ABB RAPID module: P60.mod

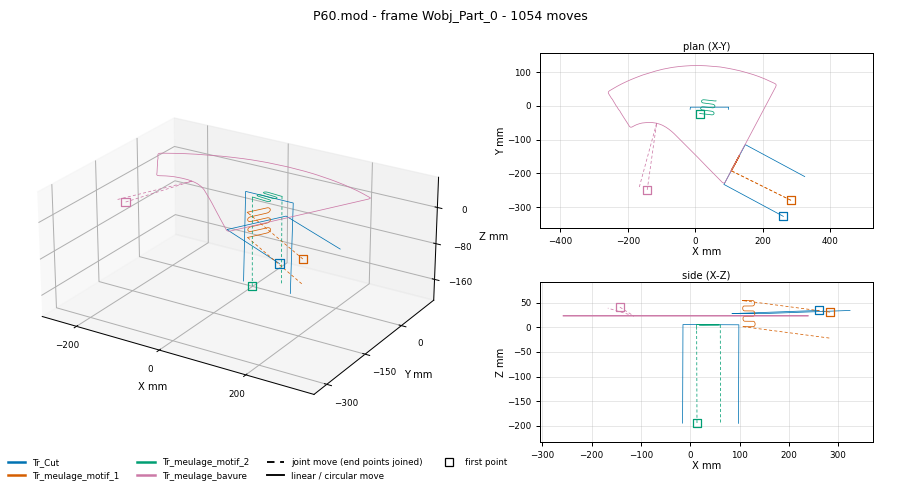
[picture p0: tool path of P60.mod in frame Wobj_Part_0, 1054 of 1064 moves have a stored position in this frame; points joined in program order, loops and branches not executed]
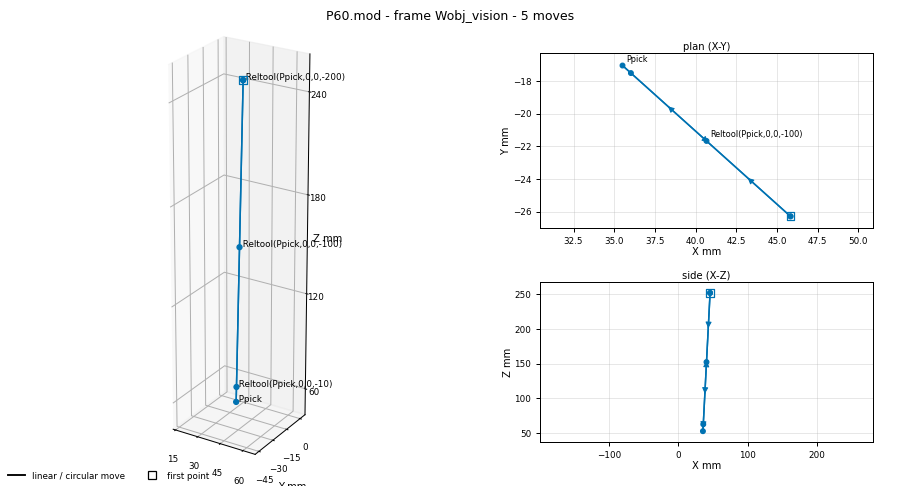
[picture p1: tool path of P60.mod in frame Wobj_vision, 5 of 1064 moves have a stored position in this frame; points joined in program order, loops and branches not executed]
MODULE P60
	LOCAL CONST Speeddata vitesse_Tronconnage :=[10, 500, 0, 0];
	LOCAL CONST Robtarget Coupe_0 :=[[118.6595,-169.366,27.637169921875],[0.183639212461518,0.161711104402732,0.6883672847491,0.682844520843884],[0,0,0,0],[8.999999E+09,8.999999E+09,8.999999E+09,8.999999E+09,8.999999E+09,8.999999E+09]];
	LOCAL CONST Robtarget Coupe_1 :=[[36.94522265625,-3.83223803710937,5.1827177734375],[0.70842525590095,-0.0115011244984384,-0.705597649362176,0.0115472140154091],[0,0,0,0],[8.999999E+09,8.999999E+09,8.999999E+09,8.999999E+09,8.999999E+09,8.999999E+09]];
	LOCAL CONST Robtarget Tr_meulage_motif_1_App1 :=[[283.559670676337,-280.003554022324,30.6185387570368],[0.635107748876336,-0.564376918949611,-0.350307497755773,0.394209966502961],[0,0,0,0],[8.999999E+09,8.999999E+09,8.999999E+09,8.999999E+09,8.999999E+09,8.999999E+09]];
	LOCAL CONST Robtarget Tr_meulage_motif_1_App2 :=[[114.472585877567,-196.272283951116,52.9486118987893],[0.635107748876336,-0.564376918949611,-0.350307497755773,0.394209966502961],[0,0,0,0],[8.999999E+09,8.999999E+09,8.999999E+09,8.999999E+09,8.999999E+09,8.999999E+09]];
	LOCAL CONST Robtarget Tr_meulage_motif_1_P0 :=[[105.573265625,-191.865375,54.12387890625],[0.635107748876336,-0.564376918949611,-0.350307497755773,0.394209966502961],[0,0,0,0],[8.999999E+09,8.999999E+09,8.999999E+09,8.999999E+09,8.999999E+09,8.999999E+09]];
	LOCAL CONST Robtarget Tr_meulage_motif_1_P1 :=[[106.0475625,-190.985015625,54.12386328125],[0.635107748876336,-0.564376918949611,-0.350307497755773,0.394209966502961],[0,0,0,0],[8.999999E+09,8.999999E+09,8.999999E+09,8.999999E+09,8.999999E+09,8.999999E+09]];
	LOCAL CONST Robtarget Tr_meulage_motif_1_P2 :=[[106.5218515625,-190.104640625,54.1238515625],[0.635107748876336,-0.564376918949611,-0.350307497755773,0.394209966502961],[0,0,0,0],[8.999999E+09,8.999999E+09,8.999999E+09,8.999999E+09,8.999999E+09,8.999999E+09]];
	LOCAL CONST Robtarget Tr_meulage_motif_1_P3 :=[[106.9961484375,-189.22428125,54.12383984375],[0.635107748876336,-0.564376918949611,-0.350307497755773,0.394209966502961],[0,0,0,0],[8.999999E+09,8.999999E+09,8.999999E+09,8.999999E+09,8.999999E+09,8.999999E+09]];
	LOCAL CONST Robtarget Tr_meulage_motif_1_P4 :=[[107.4704375,-188.34390625,54.123828125],[0.635107748876336,-0.564376918949611,-0.350307497755773,0.394209966502961],[0,0,0,0],[8.999999E+09,8.999999E+09,8.999999E+09,8.999999E+09,8.999999E+09,8.999999E+09]];
	LOCAL CONST Robtarget Tr_meulage_motif_1_P5 :=[[107.944734375,-187.463546875,54.12381640625],[0.635107748876336,-0.564376918949611,-0.350307497755773,0.394209966502961],[0,0,0,0],[8.999999E+09,8.999999E+09,8.999999E+09,8.999999E+09,8.999999E+09,8.999999E+09]];
	LOCAL CONST Robtarget Tr_meulage_motif_1_P6 :=[[108.4190234375,-186.583171875,54.1238046875],[0.635107748876336,-0.564376918949611,-0.350307497755773,0.394209966502961],[0,0,0,0],[8.999999E+09,8.999999E+09,8.999999E+09,8.999999E+09,8.999999E+09,8.999999E+09]];
	LOCAL CONST Robtarget Tr_meulage_motif_1_P7 :=[[108.8933125,-185.7028125,54.1237890625],[0.635107748876336,-0.564376918949611,-0.350307497755773,0.394209966502961],[0,0,0,0],[8.999999E+09,8.999999E+09,8.999999E+09,8.999999E+09,8.999999E+09,8.999999E+09]];
	LOCAL CONST Robtarget Tr_meulage_motif_1_P8 :=[[109.367609375,-184.8224375,54.12377734375],[0.635107748876336,-0.564376918949611,-0.350307497755773,0.394209966502961],[0,0,0,0],[8.999999E+09,8.999999E+09,8.999999E+09,8.999999E+09,8.999999E+09,8.999999E+09]];
	LOCAL CONST Robtarget Tr_meulage_motif_1_P9 :=[[109.8418984375,-183.942078125,54.123765625],[0.635107748876336,-0.564376918949611,-0.350307497755773,0.394209966502961],[0,0,0,0],[8.999999E+09,8.999999E+09,8.999999E+09,8.999999E+09,8.999999E+09,8.999999E+09]];
	LOCAL CONST Robtarget Tr_meulage_motif_1_P10 :=[[110.3161953125,-183.061703125,54.12375390625],[0.635107748876336,-0.564376918949611,-0.350307497755773,0.394209966502961],[0,0,0,0],[8.999999E+09,8.999999E+09,8.999999E+09,8.999999E+09,8.999999E+09,8.999999E+09]];
	LOCAL CONST Robtarget Tr_meulage_motif_1_P11 :=[[110.790484375,-182.18134375,54.1237421875],[0.635107748876336,-0.564376918949611,-0.350307497755773,0.394209966502961],[0,0,0,0],[8.999999E+09,8.999999E+09,8.999999E+09,8.999999E+09,8.999999E+09,8.999999E+09]];
	LOCAL CONST Robtarget Tr_meulage_motif_1_P12 :=[[111.26478125,-181.30096875,54.1237265625],[0.635107748876336,-0.564376918949611,-0.350307497755773,0.394209966502961],[0,0,0,0],[8.999999E+09,8.999999E+09,8.999999E+09,8.999999E+09,8.999999E+09,8.999999E+09]];
	LOCAL CONST Robtarget Tr_meulage_motif_1_P13 :=[[111.7390703125,-180.420609375,54.12371484375],[0.635107748876336,-0.564376918949611,-0.350307497755773,0.394209966502961],[0,0,0,0],[8.999999E+09,8.999999E+09,8.999999E+09,8.999999E+09,8.999999E+09,8.999999E+09]];
	LOCAL CONST Robtarget Tr_meulage_motif_1_P14 :=[[112.2133671875,-179.540234375,54.123703125],[0.635107748876336,-0.564376918949611,-0.350307497755773,0.394209966502961],[0,0,0,0],[8.999999E+09,8.999999E+09,8.999999E+09,8.999999E+09,8.999999E+09,8.999999E+09]];
	LOCAL CONST Robtarget Tr_meulage_motif_1_P15 :=[[112.68765625,-178.659875,54.12369140625],[0.635107748876336,-0.564376918949611,-0.350307497755773,0.394209966502961],[0,0,0,0],[8.999999E+09,8.999999E+09,8.999999E+09,8.999999E+09,8.999999E+09,8.999999E+09]];
	LOCAL CONST Robtarget Tr_meulage_motif_1_P16 :=[[113.161953125,-177.7795,54.1236796875],[0.635107748876336,-0.564376918949611,-0.350307497755773,0.394209966502961],[0,0,0,0],[8.999999E+09,8.999999E+09,8.999999E+09,8.999999E+09,8.999999E+09,8.999999E+09]];
	LOCAL CONST Robtarget Tr_meulage_motif_1_P17 :=[[113.6362421875,-176.899140625,54.1236640625],[0.635107748876336,-0.564376918949611,-0.350307497755773,0.394209966502961],[0,0,0,0],[8.999999E+09,8.999999E+09,8.999999E+09,8.999999E+09,8.999999E+09,8.999999E+09]];
	LOCAL CONST Robtarget Tr_meulage_motif_1_P18 :=[[114.1105390625,-176.018765625,54.12365234375],[0.635107748876336,-0.564376918949611,-0.350307497755773,0.394209966502961],[0,0,0,0],[8.999999E+09,8.999999E+09,8.999999E+09,8.999999E+09,8.999999E+09,8.999999E+09]];
	LOCAL CONST Robtarget Tr_meulage_motif_1_P19 :=[[114.584828125,-175.13840625,54.123640625],[0.635107748876336,-0.564376918949611,-0.350307497755773,0.394209966502961],[0,0,0,0],[8.999999E+09,8.999999E+09,8.999999E+09,8.999999E+09,8.999999E+09,8.999999E+09]];
	LOCAL CONST Robtarget Tr_meulage_motif_1_P20 :=[[115.059125,-174.25803125,54.12362890625],[0.635107748876336,-0.564376918949611,-0.350307497755773,0.394209966502961],[0,0,0,0],[8.999999E+09,8.999999E+09,8.999999E+09,8.999999E+09,8.999999E+09,8.999999E+09]];
	LOCAL CONST Robtarget Tr_meulage_motif_1_P21 :=[[115.5334140625,-173.377671875,54.1236171875],[0.635107748876336,-0.564376918949611,-0.350307497755773,0.394209966502961],[0,0,0,0],[8.999999E+09,8.999999E+09,8.999999E+09,8.999999E+09,8.999999E+09,8.999999E+09]];
	LOCAL CONST Robtarget Tr_meulage_motif_1_P22 :=[[116.0077109375,-172.497296875,54.12360546875],[0.635107748876336,-0.564376918949611,-0.350307497755773,0.394209966502961],[0,0,0,0],[8.999999E+09,8.999999E+09,8.999999E+09,8.999999E+09,8.999999E+09,8.999999E+09]];
	LOCAL CONST Robtarget Tr_meulage_motif_1_P23 :=[[116.482,-171.6169375,54.12358984375],[0.635107748876336,-0.564376918949611,-0.350307497755773,0.394209966502961],[0,0,0,0],[8.999999E+09,8.999999E+09,8.999999E+09,8.999999E+09,8.999999E+09,8.999999E+09]];
	LOCAL CONST Robtarget Tr_meulage_motif_1_P24 :=[[116.956296875,-170.7365625,54.123578125],[0.635107748876336,-0.564376918949611,-0.350307497755773,0.394209966502961],[0,0,0,0],[8.999999E+09,8.999999E+09,8.999999E+09,8.999999E+09,8.999999E+09,8.999999E+09]];
	LOCAL CONST Robtarget Tr_meulage_motif_1_P25 :=[[117.4305859375,-169.856203125,54.12356640625],[0.635107748876336,-0.564376918949611,-0.350307497755773,0.394209966502961],[0,0,0,0],[8.999999E+09,8.999999E+09,8.999999E+09,8.999999E+09,8.999999E+09,8.999999E+09]];
	LOCAL CONST Robtarget Tr_meulage_motif_1_P26 :=[[117.9048828125,-168.975828125,54.1235546875],[0.635107748876336,-0.564376918949611,-0.350307497755773,0.394209966502961],[0,0,0,0],[8.999999E+09,8.999999E+09,8.999999E+09,8.999999E+09,8.999999E+09,8.999999E+09]];
	LOCAL CONST Robtarget Tr_meulage_motif_1_P27 :=[[118.379171875,-168.09546875,54.12354296875],[0.635107748876336,-0.564376918949611,-0.350307497755773,0.394209966502961],[0,0,0,0],[8.999999E+09,8.999999E+09,8.999999E+09,8.999999E+09,8.999999E+09,8.999999E+09]];
	LOCAL CONST Robtarget Tr_meulage_motif_1_P28 :=[[118.8534609375,-167.21509375,54.12352734375],[0.635107748876336,-0.564376918949611,-0.350307497755773,0.394209966502961],[0,0,0,0],[8.999999E+09,8.999999E+09,8.999999E+09,8.999999E+09,8.999999E+09,8.999999E+09]];
	LOCAL CONST Robtarget Tr_meulage_motif_1_P29 :=[[119.3277578125,-166.334734375,54.123515625],[0.635107748876336,-0.564376918949611,-0.350307497755773,0.394209966502961],[0,0,0,0],[8.999999E+09,8.999999E+09,8.999999E+09,8.999999E+09,8.999999E+09,8.999999E+09]];
	LOCAL CONST Robtarget Tr_meulage_motif_1_P30 :=[[119.802046875,-165.454359375,54.12350390625],[0.635107748876336,-0.564376918949611,-0.350307497755773,0.394209966502961],[0,0,0,0],[8.999999E+09,8.999999E+09,8.999999E+09,8.999999E+09,8.999999E+09,8.999999E+09]];
	LOCAL CONST Robtarget Tr_meulage_motif_1_P31 :=[[120.27634375,-164.574,54.1234921875],[0.635107748876336,-0.564376918949611,-0.350307497755773,0.394209966502961],[0,0,0,0],[8.999999E+09,8.999999E+09,8.999999E+09,8.999999E+09,8.999999E+09,8.999999E+09]];
	LOCAL CONST Robtarget Tr_meulage_motif_1_P32 :=[[120.7506328125,-163.693625,54.12348046875],[0.635107748876336,-0.564376918949611,-0.350307497755773,0.394209966502961],[0,0,0,0],[8.999999E+09,8.999999E+09,8.999999E+09,8.999999E+09,8.999999E+09,8.999999E+09]];
	LOCAL CONST Robtarget Tr_meulage_motif_1_P33 :=[[121.2249296875,-162.813265625,54.12346484375],[0.635107748876336,-0.564376918949611,-0.350307497755773,0.394209966502961],[0,0,0,0],[8.999999E+09,8.999999E+09,8.999999E+09,8.999999E+09,8.999999E+09,8.999999E+09]];
	LOCAL CONST Robtarget Tr_meulage_motif_1_P34 :=[[121.69921875,-161.932890625,54.123453125],[0.635107748876336,-0.564376918949611,-0.350307497755773,0.394209966502961],[0,0,0,0],[8.999999E+09,8.999999E+09,8.999999E+09,8.999999E+09,8.999999E+09,8.999999E+09]];
	LOCAL CONST Robtarget Tr_meulage_motif_1_P35 :=[[122.173515625,-161.05253125,54.12344140625],[0.635107748876336,-0.564376918949611,-0.350307497755773,0.394209966502961],[0,0,0,0],[8.999999E+09,8.999999E+09,8.999999E+09,8.999999E+09,8.999999E+09,8.999999E+09]];
	LOCAL CONST Robtarget Tr_meulage_motif_1_P36 :=[[122.6478046875,-160.17215625,54.1234296875],[0.635107748876336,-0.564376918949611,-0.350307497755773,0.394209966502961],[0,0,0,0],[8.999999E+09,8.999999E+09,8.999999E+09,8.999999E+09,8.999999E+09,8.999999E+09]];
	LOCAL CONST Robtarget Tr_meulage_motif_1_P37 :=[[123.1221015625,-159.291796875,54.12341796875],[0.635107748876336,-0.564376918949611,-0.350307497755773,0.394209966502961],[0,0,0,0],[8.999999E+09,8.999999E+09,8.999999E+09,8.999999E+09,8.999999E+09,8.999999E+09]];
	LOCAL CONST Robtarget Tr_meulage_motif_1_P38 :=[[123.596390625,-158.411421875,54.12340625],[0.635107748876336,-0.564376918949611,-0.350307497755773,0.394209966502961],[0,0,0,0],[8.999999E+09,8.999999E+09,8.999999E+09,8.999999E+09,8.999999E+09,8.999999E+09]];
	LOCAL CONST Robtarget Tr_meulage_motif_1_P39 :=[[124.0706875,-157.5310625,54.123390625],[0.635107748876336,-0.564376918949611,-0.350307497755773,0.394209966502961],[0,0,0,0],[8.999999E+09,8.999999E+09,8.999999E+09,8.999999E+09,8.999999E+09,8.999999E+09]];
	LOCAL CONST Robtarget Tr_meulage_motif_1_P40 :=[[124.5449765625,-156.6506875,54.12337890625],[0.635107748876336,-0.564376918949611,-0.350307497755773,0.394209966502961],[0,0,0,0],[8.999999E+09,8.999999E+09,8.999999E+09,8.999999E+09,8.999999E+09,8.999999E+09]];
	LOCAL CONST Robtarget Tr_meulage_motif_1_P41 :=[[125.0192734375,-155.770328125,54.1233671875],[0.635107748876336,-0.564376918949611,-0.350307497755773,0.394209966502961],[0,0,0,0],[8.999999E+09,8.999999E+09,8.999999E+09,8.999999E+09,8.999999E+09,8.999999E+09]];
	LOCAL CONST Robtarget Tr_meulage_motif_1_P42 :=[[125.4935625,-154.889953125,54.12335546875],[0.635107748876336,-0.564376918949611,-0.350307497755773,0.394209966502961],[0,0,0,0],[8.999999E+09,8.999999E+09,8.999999E+09,8.999999E+09,8.999999E+09,8.999999E+09]];
	LOCAL CONST Robtarget Tr_meulage_motif_1_P43 :=[[125.967859375,-154.00959375,54.12334375],[0.635107748876336,-0.564376918949611,-0.350307497755773,0.394209966502961],[0,0,0,0],[8.999999E+09,8.999999E+09,8.999999E+09,8.999999E+09,8.999999E+09,8.999999E+09]];
	LOCAL CONST Robtarget Tr_meulage_motif_1_P44 :=[[126.4421484375,-153.12921875,54.123328125],[0.635107748876336,-0.564376918949611,-0.350307497755773,0.394209966502961],[0,0,0,0],[8.999999E+09,8.999999E+09,8.999999E+09,8.999999E+09,8.999999E+09,8.999999E+09]];
	LOCAL CONST Robtarget Tr_meulage_motif_1_P45 :=[[126.9164453125,-152.248859375,54.12331640625],[0.635107748876336,-0.564376918949611,-0.350307497755773,0.394209966502961],[0,0,0,0],[8.999999E+09,8.999999E+09,8.999999E+09,8.999999E+09,8.999999E+09,8.999999E+09]];
	LOCAL CONST Robtarget Tr_meulage_motif_1_P46 :=[[127.390328125,-151.37671875,54.01276953125],[0.635107748876336,-0.564376918949611,-0.350307497755773,0.394209966502961],[0,0,0,0],[8.999999E+09,8.999999E+09,8.999999E+09,8.999999E+09,8.999999E+09,8.999999E+09]];
	LOCAL CONST Robtarget Tr_meulage_motif_1_P47 :=[[127.845203125,-150.546671875,53.80167578125],[0.635107748876336,-0.564376918949611,-0.350307497755773,0.394209966502961],[0,0,0,0],[8.999999E+09,8.999999E+09,8.999999E+09,8.999999E+09,8.999999E+09,8.999999E+09]];
	LOCAL CONST Robtarget Tr_meulage_motif_1_P48 :=[[128.2573125,-149.80009375,53.5299609375],[0.635107748876336,-0.564376918949611,-0.350307497755773,0.394209966502961],[0,0,0,0],[8.999999E+09,8.999999E+09,8.999999E+09,8.999999E+09,8.999999E+09,8.999999E+09]];
	LOCAL CONST Robtarget Tr_meulage_motif_1_P49 :=[[128.6207890625,-149.144078125,53.25415625],[0.635107748876336,-0.564376918949611,-0.350307497755773,0.394209966502961],[0,0,0,0],[8.999999E+09,8.999999E+09,8.999999E+09,8.999999E+09,8.999999E+09,8.999999E+09]];
	LOCAL CONST Robtarget Tr_meulage_motif_1_P50 :=[[129.160390625,-148.184109375,52.6383359375],[0.635107748876336,-0.564376918949611,-0.350307497755773,0.394209966502961],[0,0,0,0],[8.999999E+09,8.999999E+09,8.999999E+09,8.999999E+09,8.999999E+09,8.999999E+09]];
	LOCAL CONST Robtarget Tr_meulage_motif_1_P51 :=[[129.669921875,-147.295609375,51.7911015625],[0.635107748876336,-0.564376918949611,-0.350307497755773,0.394209966502961],[0,0,0,0],[8.999999E+09,8.999999E+09,8.999999E+09,8.999999E+09,8.999999E+09,8.999999E+09]];
	LOCAL CONST Robtarget Tr_meulage_motif_1_P52 :=[[130.1008515625,-146.5649375,50.7677421875],[0.635107748876336,-0.564376918949611,-0.350307497755773,0.394209966502961],[0,0,0,0],[8.999999E+09,8.999999E+09,8.999999E+09,8.999999E+09,8.999999E+09,8.999999E+09]];
	LOCAL CONST Robtarget Tr_meulage_motif_1_P53 :=[[130.3638671875,-146.152171875,49.65212109375],[0.635107748876336,-0.564376918949611,-0.350307497755773,0.394209966502961],[0,0,0,0],[8.999999E+09,8.999999E+09,8.999999E+09,8.999999E+09,8.999999E+09,8.999999E+09]];
	LOCAL CONST Robtarget Tr_meulage_motif_1_P54 :=[[130.3963359375,-146.1389375,48.95651171875],[0.635107748876336,-0.564376918949611,-0.350307497755773,0.394209966502961],[0,0,0,0],[8.999999E+09,8.999999E+09,8.999999E+09,8.999999E+09,8.999999E+09,8.999999E+09]];
	LOCAL CONST Robtarget Tr_meulage_motif_1_P55 :=[[130.4149921875,-146.148984375,48.2956015625],[0.635107748876336,-0.564376918949611,-0.350307497755773,0.394209966502961],[0,0,0,0],[8.999999E+09,8.999999E+09,8.999999E+09,8.999999E+09,8.999999E+09,8.999999E+09]];
	LOCAL CONST Robtarget Tr_meulage_motif_1_P56 :=[[130.4076171875,-146.207359375,47.63484765625],[0.635107748876336,-0.564376918949611,-0.350307497755773,0.394209966502961],[0,0,0,0],[8.999999E+09,8.999999E+09,8.999999E+09,8.999999E+09,8.999999E+09,8.999999E+09]];
	LOCAL CONST Robtarget Tr_meulage_motif_1_P57 :=[[130.2023984375,-146.662734375,46.53366796875],[0.635107748876336,-0.564376918949611,-0.350307497755773,0.394209966502961],[0,0,0,0],[8.999999E+09,8.999999E+09,8.999999E+09,8.999999E+09,8.999999E+09,8.999999E+09]];
	LOCAL CONST Robtarget Tr_meulage_motif_1_P58 :=[[129.8245078125,-147.4321875,45.52757421875],[0.635107748876336,-0.564376918949611,-0.350307497755773,0.394209966502961],[0,0,0,0],[8.999999E+09,8.999999E+09,8.999999E+09,8.999999E+09,8.999999E+09,8.999999E+09]];
	LOCAL CONST Robtarget Tr_meulage_motif_1_P59 :=[[129.3625,-148.34578125,44.69913671875],[0.635107748876336,-0.564376918949611,-0.350307497755773,0.394209966502961],[0,0,0,0],[8.999999E+09,8.999999E+09,8.999999E+09,8.999999E+09,8.999999E+09,8.999999E+09]];
	LOCAL CONST Robtarget Tr_meulage_motif_1_P60 :=[[129.04778125,-148.9566875,44.30359765625],[0.635107748876336,-0.564376918949611,-0.350307497755773,0.394209966502961],[0,0,0,0],[8.999999E+09,8.999999E+09,8.999999E+09,8.999999E+09,8.999999E+09,8.999999E+09]];
	LOCAL CONST Robtarget Tr_meulage_motif_1_P61 :=[[128.5122265625,-149.98371875,43.81633203125],[0.635107748876336,-0.564376918949611,-0.350307497755773,0.394209966502961],[0,0,0,0],[8.999999E+09,8.999999E+09,8.999999E+09,8.999999E+09,8.999999E+09,8.999999E+09]];
	LOCAL CONST Robtarget Tr_meulage_motif_1_P62 :=[[128.1188828125,-150.731671875,43.5523828125],[0.635107748876336,-0.564376918949611,-0.350307497755773,0.394209966502961],[0,0,0,0],[8.999999E+09,8.999999E+09,8.999999E+09,8.999999E+09,8.999999E+09,8.999999E+09]];
	LOCAL CONST Robtarget Tr_meulage_motif_1_P63 :=[[127.6826171875,-151.55528125,43.34803125],[0.635107748876336,-0.564376918949611,-0.350307497755773,0.394209966502961],[0,0,0,0],[8.999999E+09,8.999999E+09,8.999999E+09,8.999999E+09,8.999999E+09,8.999999E+09]];
	LOCAL CONST Robtarget Tr_meulage_motif_1_P64 :=[[127.2201328125,-152.4210625,43.2395078125],[0.635107748876336,-0.564376918949611,-0.350307497755773,0.394209966502961],[0,0,0,0],[8.999999E+09,8.999999E+09,8.999999E+09,8.999999E+09,8.999999E+09,8.999999E+09]];
	LOCAL CONST Robtarget Tr_meulage_motif_1_P65 :=[[126.752484375,-153.2965625,43.12898046875],[0.635107748876336,-0.564376918949611,-0.350307497755773,0.394209966502961],[0,0,0,0],[8.999999E+09,8.999999E+09,8.999999E+09,8.999999E+09,8.999999E+09,8.999999E+09]];
	LOCAL CONST Robtarget Tr_meulage_motif_1_P66 :=[[126.2781875,-154.1769375,43.12899609375],[0.635107748876336,-0.564376918949611,-0.350307497755773,0.394209966502961],[0,0,0,0],[8.999999E+09,8.999999E+09,8.999999E+09,8.999999E+09,8.999999E+09,8.999999E+09]];
	LOCAL CONST Robtarget Tr_meulage_motif_1_P67 :=[[125.8038984375,-155.057296875,43.1290078125],[0.635107748876336,-0.564376918949611,-0.350307497755773,0.394209966502961],[0,0,0,0],[8.999999E+09,8.999999E+09,8.999999E+09,8.999999E+09,8.999999E+09,8.999999E+09]];
	LOCAL CONST Robtarget Tr_meulage_motif_1_P68 :=[[125.329609375,-155.937671875,43.12901953125],[0.635107748876336,-0.564376918949611,-0.350307497755773,0.394209966502961],[0,0,0,0],[8.999999E+09,8.999999E+09,8.999999E+09,8.999999E+09,8.999999E+09,8.999999E+09]];
	LOCAL CONST Robtarget Tr_meulage_motif_1_P69 :=[[124.8553125,-156.81803125,43.12903125],[0.635107748876336,-0.564376918949611,-0.350307497755773,0.394209966502961],[0,0,0,0],[8.999999E+09,8.999999E+09,8.999999E+09,8.999999E+09,8.999999E+09,8.999999E+09]];
	LOCAL CONST Robtarget Tr_meulage_motif_1_P70 :=[[124.3810234375,-157.69840625,43.12904296875],[0.635107748876336,-0.564376918949611,-0.350307497755773,0.394209966502961],[0,0,0,0],[8.999999E+09,8.999999E+09,8.999999E+09,8.999999E+09,8.999999E+09,8.999999E+09]];
	LOCAL CONST Robtarget Tr_meulage_motif_1_P71 :=[[123.9067265625,-158.578765625,43.1290546875],[0.635107748876336,-0.564376918949611,-0.350307497755773,0.394209966502961],[0,0,0,0],[8.999999E+09,8.999999E+09,8.999999E+09,8.999999E+09,8.999999E+09,8.999999E+09]];
	LOCAL CONST Robtarget Tr_meulage_motif_1_P72 :=[[123.4324375,-159.459140625,43.1290703125],[0.635107748876336,-0.564376918949611,-0.350307497755773,0.394209966502961],[0,0,0,0],[8.999999E+09,8.999999E+09,8.999999E+09,8.999999E+09,8.999999E+09,8.999999E+09]];
	LOCAL CONST Robtarget Tr_meulage_motif_1_P73 :=[[122.958140625,-160.3395,43.12908203125],[0.635107748876336,-0.564376918949611,-0.350307497755773,0.394209966502961],[0,0,0,0],[8.999999E+09,8.999999E+09,8.999999E+09,8.999999E+09,8.999999E+09,8.999999E+09]];
	LOCAL CONST Robtarget Tr_meulage_motif_1_P74 :=[[122.4838515625,-161.219875,43.12909375],[0.635107748876336,-0.564376918949611,-0.350307497755773,0.394209966502961],[0,0,0,0],[8.999999E+09,8.999999E+09,8.999999E+09,8.999999E+09,8.999999E+09,8.999999E+09]];
	LOCAL CONST Robtarget Tr_meulage_motif_1_P75 :=[[122.0095546875,-162.100234375,43.12910546875],[0.635107748876336,-0.564376918949611,-0.350307497755773,0.394209966502961],[0,0,0,0],[8.999999E+09,8.999999E+09,8.999999E+09,8.999999E+09,8.999999E+09,8.999999E+09]];
	LOCAL CONST Robtarget Tr_meulage_motif_1_P76 :=[[121.535265625,-162.980609375,43.1291171875],[0.635107748876336,-0.564376918949611,-0.350307497755773,0.394209966502961],[0,0,0,0],[8.999999E+09,8.999999E+09,8.999999E+09,8.999999E+09,8.999999E+09,8.999999E+09]];
	LOCAL CONST Robtarget Tr_meulage_motif_1_P77 :=[[121.06096875,-163.86096875,43.1291328125],[0.635107748876336,-0.564376918949611,-0.350307497755773,0.394209966502961],[0,0,0,0],[8.999999E+09,8.999999E+09,8.999999E+09,8.999999E+09,8.999999E+09,8.999999E+09]];
	LOCAL CONST Robtarget Tr_meulage_motif_1_P78 :=[[120.5866796875,-164.74134375,43.12914453125],[0.635107748876336,-0.564376918949611,-0.350307497755773,0.394209966502961],[0,0,0,0],[8.999999E+09,8.999999E+09,8.999999E+09,8.999999E+09,8.999999E+09,8.999999E+09]];
	LOCAL CONST Robtarget Tr_meulage_motif_1_P79 :=[[120.1123828125,-165.621703125,43.12915625],[0.635107748876336,-0.564376918949611,-0.350307497755773,0.394209966502961],[0,0,0,0],[8.999999E+09,8.999999E+09,8.999999E+09,8.999999E+09,8.999999E+09,8.999999E+09]];
	LOCAL CONST Robtarget Tr_meulage_motif_1_P80 :=[[119.63809375,-166.502078125,43.12916796875],[0.635107748876336,-0.564376918949611,-0.350307497755773,0.394209966502961],[0,0,0,0],[8.999999E+09,8.999999E+09,8.999999E+09,8.999999E+09,8.999999E+09,8.999999E+09]];
	LOCAL CONST Robtarget Tr_meulage_motif_1_P81 :=[[119.163796875,-167.3824375,43.1291796875],[0.635107748876336,-0.564376918949611,-0.350307497755773,0.394209966502961],[0,0,0,0],[8.999999E+09,8.999999E+09,8.999999E+09,8.999999E+09,8.999999E+09,8.999999E+09]];
	LOCAL CONST Robtarget Tr_meulage_motif_1_P82 :=[[118.6895078125,-168.2628125,43.1291953125],[0.635107748876336,-0.564376918949611,-0.350307497755773,0.394209966502961],[0,0,0,0],[8.999999E+09,8.999999E+09,8.999999E+09,8.999999E+09,8.999999E+09,8.999999E+09]];
	LOCAL CONST Robtarget Tr_meulage_motif_1_P83 :=[[118.2152109375,-169.143171875,43.12920703125],[0.635107748876336,-0.564376918949611,-0.350307497755773,0.394209966502961],[0,0,0,0],[8.999999E+09,8.999999E+09,8.999999E+09,8.999999E+09,8.999999E+09,8.999999E+09]];
	LOCAL CONST Robtarget Tr_meulage_motif_1_P84 :=[[117.740921875,-170.023546875,43.12921875],[0.635107748876336,-0.564376918949611,-0.350307497755773,0.394209966502961],[0,0,0,0],[8.999999E+09,8.999999E+09,8.999999E+09,8.999999E+09,8.999999E+09,8.999999E+09]];
	LOCAL CONST Robtarget Tr_meulage_motif_1_P85 :=[[117.266625,-170.90390625,43.12923046875],[0.635107748876336,-0.564376918949611,-0.350307497755773,0.394209966502961],[0,0,0,0],[8.999999E+09,8.999999E+09,8.999999E+09,8.999999E+09,8.999999E+09,8.999999E+09]];
	LOCAL CONST Robtarget Tr_meulage_motif_1_P86 :=[[116.7923359375,-171.78428125,43.1292421875],[0.635107748876336,-0.564376918949611,-0.350307497755773,0.394209966502961],[0,0,0,0],[8.999999E+09,8.999999E+09,8.999999E+09,8.999999E+09,8.999999E+09,8.999999E+09]];
	LOCAL CONST Robtarget Tr_meulage_motif_1_P87 :=[[116.3180390625,-172.664640625,43.12925390625],[0.635107748876336,-0.564376918949611,-0.350307497755773,0.394209966502961],[0,0,0,0],[8.999999E+09,8.999999E+09,8.999999E+09,8.999999E+09,8.999999E+09,8.999999E+09]];
	LOCAL CONST Robtarget Tr_meulage_motif_1_P88 :=[[115.84375,-173.545015625,43.12926953125],[0.635107748876336,-0.564376918949611,-0.350307497755773,0.394209966502961],[0,0,0,0],[8.999999E+09,8.999999E+09,8.999999E+09,8.999999E+09,8.999999E+09,8.999999E+09]];
	LOCAL CONST Robtarget Tr_meulage_motif_1_P89 :=[[115.3694609375,-174.425375,43.12928125],[0.635107748876336,-0.564376918949611,-0.350307497755773,0.394209966502961],[0,0,0,0],[8.999999E+09,8.999999E+09,8.999999E+09,8.999999E+09,8.999999E+09,8.999999E+09]];
	LOCAL CONST Robtarget Tr_meulage_motif_1_P90 :=[[114.8951640625,-175.30575,43.12929296875],[0.635107748876336,-0.564376918949611,-0.350307497755773,0.394209966502961],[0,0,0,0],[8.999999E+09,8.999999E+09,8.999999E+09,8.999999E+09,8.999999E+09,8.999999E+09]];
	LOCAL CONST Robtarget Tr_meulage_motif_1_P91 :=[[114.420875,-176.186109375,43.1293046875],[0.635107748876336,-0.564376918949611,-0.350307497755773,0.394209966502961],[0,0,0,0],[8.999999E+09,8.999999E+09,8.999999E+09,8.999999E+09,8.999999E+09,8.999999E+09]];
	LOCAL CONST Robtarget Tr_meulage_motif_1_P92 :=[[113.946578125,-177.066484375,43.12931640625],[0.635107748876336,-0.564376918949611,-0.350307497755773,0.394209966502961],[0,0,0,0],[8.999999E+09,8.999999E+09,8.999999E+09,8.999999E+09,8.999999E+09,8.999999E+09]];
	LOCAL CONST Robtarget Tr_meulage_motif_1_P93 :=[[113.4722890625,-177.94684375,43.12933203125],[0.635107748876336,-0.564376918949611,-0.350307497755773,0.394209966502961],[0,0,0,0],[8.999999E+09,8.999999E+09,8.999999E+09,8.999999E+09,8.999999E+09,8.999999E+09]];
	LOCAL CONST Robtarget Tr_meulage_motif_1_P94 :=[[112.9979921875,-178.82721875,43.12934375],[0.635107748876336,-0.564376918949611,-0.350307497755773,0.394209966502961],[0,0,0,0],[8.999999E+09,8.999999E+09,8.999999E+09,8.999999E+09,8.999999E+09,8.999999E+09]];
	LOCAL CONST Robtarget Tr_meulage_motif_1_P95 :=[[112.523703125,-179.707578125,43.12935546875],[0.635107748876336,-0.564376918949611,-0.350307497755773,0.394209966502961],[0,0,0,0],[8.999999E+09,8.999999E+09,8.999999E+09,8.999999E+09,8.999999E+09,8.999999E+09]];
	LOCAL CONST Robtarget Tr_meulage_motif_1_P96 :=[[112.04940625,-180.587953125,43.1293671875],[0.635107748876336,-0.564376918949611,-0.350307497755773,0.394209966502961],[0,0,0,0],[8.999999E+09,8.999999E+09,8.999999E+09,8.999999E+09,8.999999E+09,8.999999E+09]];
	LOCAL CONST Robtarget Tr_meulage_motif_1_P97 :=[[111.5751171875,-181.4683125,43.12937890625],[0.635107748876336,-0.564376918949611,-0.350307497755773,0.394209966502961],[0,0,0,0],[8.999999E+09,8.999999E+09,8.999999E+09,8.999999E+09,8.999999E+09,8.999999E+09]];
	LOCAL CONST Robtarget Tr_meulage_motif_1_P98 :=[[111.1008203125,-182.3486875,43.12939453125],[0.635107748876336,-0.564376918949611,-0.350307497755773,0.394209966502961],[0,0,0,0],[8.999999E+09,8.999999E+09,8.999999E+09,8.999999E+09,8.999999E+09,8.999999E+09]];
	LOCAL CONST Robtarget Tr_meulage_motif_1_P99 :=[[110.62653125,-183.229046875,43.12940625],[0.635107748876336,-0.564376918949611,-0.350307497755773,0.394209966502961],[0,0,0,0],[8.999999E+09,8.999999E+09,8.999999E+09,8.999999E+09,8.999999E+09,8.999999E+09]];
	LOCAL CONST Robtarget Tr_meulage_motif_1_P100 :=[[110.152234375,-184.109421875,43.12941796875],[0.635107748876336,-0.564376918949611,-0.350307497755773,0.394209966502961],[0,0,0,0],[8.999999E+09,8.999999E+09,8.999999E+09,8.999999E+09,8.999999E+09,8.999999E+09]];
	LOCAL CONST Robtarget Tr_meulage_motif_1_P101 :=[[109.6779453125,-184.98978125,43.1294296875],[0.635107748876336,-0.564376918949611,-0.350307497755773,0.394209966502961],[0,0,0,0],[8.999999E+09,8.999999E+09,8.999999E+09,8.999999E+09,8.999999E+09,8.999999E+09]];
	LOCAL CONST Robtarget Tr_meulage_motif_1_P102 :=[[109.2036484375,-185.87015625,43.12944140625],[0.635107748876336,-0.564376918949611,-0.350307497755773,0.394209966502961],[0,0,0,0],[8.999999E+09,8.999999E+09,8.999999E+09,8.999999E+09,8.999999E+09,8.999999E+09]];
	LOCAL CONST Robtarget Tr_meulage_motif_1_P103 :=[[108.7360078125,-186.74565625,43.01891796875],[0.635107748876336,-0.564376918949611,-0.350307497755773,0.394209966502961],[0,0,0,0],[8.999999E+09,8.999999E+09,8.999999E+09,8.999999E+09,8.999999E+09,8.999999E+09]];
	LOCAL CONST Robtarget Tr_meulage_motif_1_P104 :=[[108.293046875,-187.582140625,42.8078515625],[0.635107748876336,-0.564376918949611,-0.350307497755773,0.394209966502961],[0,0,0,0],[8.999999E+09,8.999999E+09,8.999999E+09,8.999999E+09,8.999999E+09,8.999999E+09]];
	LOCAL CONST Robtarget Tr_meulage_motif_1_P105 :=[[107.8962734375,-188.336984375,42.53615625],[0.635107748876336,-0.564376918949611,-0.350307497755773,0.394209966502961],[0,0,0,0],[8.999999E+09,8.999999E+09,8.999999E+09,8.999999E+09,8.999999E+09,8.999999E+09]];
	LOCAL CONST Robtarget Tr_meulage_motif_1_P106 :=[[107.5673984375,-188.967984375,42.23216796875],[0.635107748876336,-0.564376918949611,-0.350307497755773,0.394209966502961],[0,0,0,0],[8.999999E+09,8.999999E+09,8.999999E+09,8.999999E+09,8.999999E+09,8.999999E+09]];
	LOCAL CONST Robtarget Tr_meulage_motif_1_P107 :=[[107.0954453125,-189.88878125,41.56998828125],[0.635107748876336,-0.564376918949611,-0.350307497755773,0.394209966502961],[0,0,0,0],[8.999999E+09,8.999999E+09,8.999999E+09,8.999999E+09,8.999999E+09,8.999999E+09]];
	LOCAL CONST Robtarget Tr_meulage_motif_1_P108 :=[[106.693109375,-190.69653125,40.6685234375],[0.635107748876336,-0.564376918949611,-0.350307497755773,0.394209966502961],[0,0,0,0],[8.999999E+09,8.999999E+09,8.999999E+09,8.999999E+09,8.999999E+09,8.999999E+09]];
	LOCAL CONST Robtarget Tr_meulage_motif_1_P109 :=[[106.468890625,-191.183421875,39.6230390625],[0.635107748876336,-0.564376918949611,-0.350307497755773,0.394209966502961],[0,0,0,0],[8.999999E+09,8.999999E+09,8.999999E+09,8.999999E+09,8.999999E+09,8.999999E+09]];
	LOCAL CONST Robtarget Tr_meulage_motif_1_P110 :=[[106.4008046875,-191.356640625,38.9301796875],[0.635107748876336,-0.564376918949611,-0.350307497755773,0.394209966502961],[0,0,0,0],[8.999999E+09,8.999999E+09,8.999999E+09,8.999999E+09,8.999999E+09,8.999999E+09]];
	LOCAL CONST Robtarget Tr_meulage_motif_1_P111 :=[[106.39225,-191.4245625,38.16057421875],[0.635107748876336,-0.564376918949611,-0.350307497755773,0.394209966502961],[0,0,0,0],[8.999999E+09,8.999999E+09,8.999999E+09,8.999999E+09,8.999999E+09,8.999999E+09]];
	LOCAL CONST Robtarget Tr_meulage_motif_1_P112 :=[[106.44571875,-191.37734375,37.39109375],[0.635107748876336,-0.564376918949611,-0.350307497755773,0.394209966502961],[0,0,0,0],[8.999999E+09,8.999999E+09,8.999999E+09,8.999999E+09,8.999999E+09,8.999999E+09]];
	LOCAL CONST Robtarget Tr_meulage_motif_1_P113 :=[[106.6759921875,-191.0248125,36.28341015625],[0.635107748876336,-0.564376918949611,-0.350307497755773,0.394209966502961],[0,0,0,0],[8.999999E+09,8.999999E+09,8.999999E+09,8.999999E+09,8.999999E+09,8.999999E+09]];
	LOCAL CONST Robtarget Tr_meulage_motif_1_P114 :=[[106.8890234375,-190.66896875,35.698015625],[0.635107748876336,-0.564376918949611,-0.350307497755773,0.394209966502961],[0,0,0,0],[8.999999E+09,8.999999E+09,8.999999E+09,8.999999E+09,8.999999E+09,8.999999E+09]];
	LOCAL CONST Robtarget Tr_meulage_motif_1_P115 :=[[107.3348125,-189.90146875,34.8113359375],[0.635107748876336,-0.564376918949611,-0.350307497755773,0.394209966502961],[0,0,0,0],[8.999999E+09,8.999999E+09,8.999999E+09,8.999999E+09,8.999999E+09,8.999999E+09]];
	LOCAL CONST Robtarget Tr_meulage_motif_1_P116 :=[[107.6242890625,-189.39215625,34.39723046875],[0.635107748876336,-0.564376918949611,-0.350307497755773,0.394209966502961],[0,0,0,0],[8.999999E+09,8.999999E+09,8.999999E+09,8.999999E+09,8.999999E+09,8.999999E+09]];
	LOCAL CONST Robtarget Tr_meulage_motif_1_P117 :=[[108.1698515625,-188.416265625,33.85340234375],[0.635107748876336,-0.564376918949611,-0.350307497755773,0.394209966502961],[0,0,0,0],[8.999999E+09,8.999999E+09,8.999999E+09,8.999999E+09,8.999999E+09,8.999999E+09]];
	LOCAL CONST Robtarget Tr_meulage_motif_1_P118 :=[[108.5697578125,-187.6939375,33.55804296875],[0.635107748876336,-0.564376918949611,-0.350307497755773,0.394209966502961],[0,0,0,0],[8.999999E+09,8.999999E+09,8.999999E+09,8.999999E+09,8.999999E+09,8.999999E+09]];
	LOCAL CONST Robtarget Tr_meulage_motif_1_P119 :=[[109.0175703125,-186.876546875,33.35366796875],[0.635107748876336,-0.564376918949611,-0.350307497755773,0.394209966502961],[0,0,0,0],[8.999999E+09,8.999999E+09,8.999999E+09,8.999999E+09,8.999999E+09,8.999999E+09]];
	LOCAL CONST Robtarget Tr_meulage_motif_1_P120 :=[[109.4861796875,-186.0140625,33.2451171875],[0.635107748876336,-0.564376918949611,-0.350307497755773,0.394209966502961],[0,0,0,0],[8.999999E+09,8.999999E+09,8.999999E+09,8.999999E+09,8.999999E+09,8.999999E+09]];
	LOCAL CONST Robtarget Tr_meulage_motif_1_P121 :=[[109.9600703125,-185.141921875,33.13456640625],[0.635107748876336,-0.564376918949611,-0.350307497755773,0.394209966502961],[0,0,0,0],[8.999999E+09,8.999999E+09,8.999999E+09,8.999999E+09,8.999999E+09,8.999999E+09]];
	LOCAL CONST Robtarget Tr_meulage_motif_1_P122 :=[[110.434359375,-184.261546875,33.1345546875],[0.635107748876336,-0.564376918949611,-0.350307497755773,0.394209966502961],[0,0,0,0],[8.999999E+09,8.999999E+09,8.999999E+09,8.999999E+09,8.999999E+09,8.999999E+09]];
	LOCAL CONST Robtarget Tr_meulage_motif_1_P123 :=[[110.9086484375,-183.3811875,33.13454296875],[0.635107748876336,-0.564376918949611,-0.350307497755773,0.394209966502961],[0,0,0,0],[8.999999E+09,8.999999E+09,8.999999E+09,8.999999E+09,8.999999E+09,8.999999E+09]];
	LOCAL CONST Robtarget Tr_meulage_motif_1_P124 :=[[111.3829453125,-182.5008125,33.13453125],[0.635107748876336,-0.564376918949611,-0.350307497755773,0.394209966502961],[0,0,0,0],[8.999999E+09,8.999999E+09,8.999999E+09,8.999999E+09,8.999999E+09,8.999999E+09]];
	LOCAL CONST Robtarget Tr_meulage_motif_1_P125 :=[[111.857234375,-181.620453125,33.13451953125],[0.635107748876336,-0.564376918949611,-0.350307497755773,0.394209966502961],[0,0,0,0],[8.999999E+09,8.999999E+09,8.999999E+09,8.999999E+09,8.999999E+09,8.999999E+09]];
	LOCAL CONST Robtarget Tr_meulage_motif_1_P126 :=[[112.33153125,-180.740078125,33.1345078125],[0.635107748876336,-0.564376918949611,-0.350307497755773,0.394209966502961],[0,0,0,0],[8.999999E+09,8.999999E+09,8.999999E+09,8.999999E+09,8.999999E+09,8.999999E+09]];
	LOCAL CONST Robtarget Tr_meulage_motif_1_P127 :=[[112.8058203125,-179.85971875,33.1344921875],[0.635107748876336,-0.564376918949611,-0.350307497755773,0.394209966502961],[0,0,0,0],[8.999999E+09,8.999999E+09,8.999999E+09,8.999999E+09,8.999999E+09,8.999999E+09]];
	LOCAL CONST Robtarget Tr_meulage_motif_1_P128 :=[[113.2801171875,-178.97934375,33.13448046875],[0.635107748876336,-0.564376918949611,-0.350307497755773,0.394209966502961],[0,0,0,0],[8.999999E+09,8.999999E+09,8.999999E+09,8.999999E+09,8.999999E+09,8.999999E+09]];
	LOCAL CONST Robtarget Tr_meulage_motif_1_P129 :=[[113.75440625,-178.098984375,33.13446875],[0.635107748876336,-0.564376918949611,-0.350307497755773,0.394209966502961],[0,0,0,0],[8.999999E+09,8.999999E+09,8.999999E+09,8.999999E+09,8.999999E+09,8.999999E+09]];
	LOCAL CONST Robtarget Tr_meulage_motif_1_P130 :=[[114.228703125,-177.218609375,33.13445703125],[0.635107748876336,-0.564376918949611,-0.350307497755773,0.394209966502961],[0,0,0,0],[8.999999E+09,8.999999E+09,8.999999E+09,8.999999E+09,8.999999E+09,8.999999E+09]];
	LOCAL CONST Robtarget Tr_meulage_motif_1_P131 :=[[114.7029921875,-176.33825,33.1344453125],[0.635107748876336,-0.564376918949611,-0.350307497755773,0.394209966502961],[0,0,0,0],[8.999999E+09,8.999999E+09,8.999999E+09,8.999999E+09,8.999999E+09,8.999999E+09]];
	LOCAL CONST Robtarget Tr_meulage_motif_1_P132 :=[[115.1772890625,-175.457875,33.1344296875],[0.635107748876336,-0.564376918949611,-0.350307497755773,0.394209966502961],[0,0,0,0],[8.999999E+09,8.999999E+09,8.999999E+09,8.999999E+09,8.999999E+09,8.999999E+09]];
	LOCAL CONST Robtarget Tr_meulage_motif_1_P133 :=[[115.651578125,-174.577515625,33.13441796875],[0.635107748876336,-0.564376918949611,-0.350307497755773,0.394209966502961],[0,0,0,0],[8.999999E+09,8.999999E+09,8.999999E+09,8.999999E+09,8.999999E+09,8.999999E+09]];
	LOCAL CONST Robtarget Tr_meulage_motif_1_P134 :=[[116.125875,-173.697140625,33.13440625],[0.635107748876336,-0.564376918949611,-0.350307497755773,0.394209966502961],[0,0,0,0],[8.999999E+09,8.999999E+09,8.999999E+09,8.999999E+09,8.999999E+09,8.999999E+09]];
	LOCAL CONST Robtarget Tr_meulage_motif_1_P135 :=[[116.6001640625,-172.81678125,33.13439453125],[0.635107748876336,-0.564376918949611,-0.350307497755773,0.394209966502961],[0,0,0,0],[8.999999E+09,8.999999E+09,8.999999E+09,8.999999E+09,8.999999E+09,8.999999E+09]];
	LOCAL CONST Robtarget Tr_meulage_motif_1_P136 :=[[117.0744609375,-171.93640625,33.1343828125],[0.635107748876336,-0.564376918949611,-0.350307497755773,0.394209966502961],[0,0,0,0],[8.999999E+09,8.999999E+09,8.999999E+09,8.999999E+09,8.999999E+09,8.999999E+09]];
	LOCAL CONST Robtarget Tr_meulage_motif_1_P137 :=[[117.54875,-171.056046875,33.1343671875],[0.635107748876336,-0.564376918949611,-0.350307497755773,0.394209966502961],[0,0,0,0],[8.999999E+09,8.999999E+09,8.999999E+09,8.999999E+09,8.999999E+09,8.999999E+09]];
	LOCAL CONST Robtarget Tr_meulage_motif_1_P138 :=[[118.023046875,-170.175671875,33.13435546875],[0.635107748876336,-0.564376918949611,-0.350307497755773,0.394209966502961],[0,0,0,0],[8.999999E+09,8.999999E+09,8.999999E+09,8.999999E+09,8.999999E+09,8.999999E+09]];
	LOCAL CONST Robtarget Tr_meulage_motif_1_P139 :=[[118.4973359375,-169.2953125,33.13434375],[0.635107748876336,-0.564376918949611,-0.350307497755773,0.394209966502961],[0,0,0,0],[8.999999E+09,8.999999E+09,8.999999E+09,8.999999E+09,8.999999E+09,8.999999E+09]];
	LOCAL CONST Robtarget Tr_meulage_motif_1_P140 :=[[118.9716328125,-168.4149375,33.13433203125],[0.635107748876336,-0.564376918949611,-0.350307497755773,0.394209966502961],[0,0,0,0],[8.999999E+09,8.999999E+09,8.999999E+09,8.999999E+09,8.999999E+09,8.999999E+09]];
	LOCAL CONST Robtarget Tr_meulage_motif_1_P141 :=[[119.445921875,-167.534578125,33.1343203125],[0.635107748876336,-0.564376918949611,-0.350307497755773,0.394209966502961],[0,0,0,0],[8.999999E+09,8.999999E+09,8.999999E+09,8.999999E+09,8.999999E+09,8.999999E+09]];
	LOCAL CONST Robtarget Tr_meulage_motif_1_P142 :=[[119.92021875,-166.654203125,33.13430859375],[0.635107748876336,-0.564376918949611,-0.350307497755773,0.394209966502961],[0,0,0,0],[8.999999E+09,8.999999E+09,8.999999E+09,8.999999E+09,8.999999E+09,8.999999E+09]];
	LOCAL CONST Robtarget Tr_meulage_motif_1_P143 :=[[120.3945078125,-165.77384375,33.13429296875],[0.635107748876336,-0.564376918949611,-0.350307497755773,0.394209966502961],[0,0,0,0],[8.999999E+09,8.999999E+09,8.999999E+09,8.999999E+09,8.999999E+09,8.999999E+09]];
	LOCAL CONST Robtarget Tr_meulage_motif_1_P144 :=[[120.868796875,-164.89346875,33.13428125],[0.635107748876336,-0.564376918949611,-0.350307497755773,0.394209966502961],[0,0,0,0],[8.999999E+09,8.999999E+09,8.999999E+09,8.999999E+09,8.999999E+09,8.999999E+09]];
	LOCAL CONST Robtarget Tr_meulage_motif_1_P145 :=[[121.34309375,-164.013109375,33.13426953125],[0.635107748876336,-0.564376918949611,-0.350307497755773,0.394209966502961],[0,0,0,0],[8.999999E+09,8.999999E+09,8.999999E+09,8.999999E+09,8.999999E+09,8.999999E+09]];
	LOCAL CONST Robtarget Tr_meulage_motif_1_P146 :=[[121.8173828125,-163.132734375,33.1342578125],[0.635107748876336,-0.564376918949611,-0.350307497755773,0.394209966502961],[0,0,0,0],[8.999999E+09,8.999999E+09,8.999999E+09,8.999999E+09,8.999999E+09,8.999999E+09]];
	LOCAL CONST Robtarget Tr_meulage_motif_1_P147 :=[[122.2916796875,-162.252375,33.13424609375],[0.635107748876336,-0.564376918949611,-0.350307497755773,0.394209966502961],[0,0,0,0],[8.999999E+09,8.999999E+09,8.999999E+09,8.999999E+09,8.999999E+09,8.999999E+09]];
	LOCAL CONST Robtarget Tr_meulage_motif_1_P148 :=[[122.76596875,-161.372,33.13423046875],[0.635107748876336,-0.564376918949611,-0.350307497755773,0.394209966502961],[0,0,0,0],[8.999999E+09,8.999999E+09,8.999999E+09,8.999999E+09,8.999999E+09,8.999999E+09]];
	LOCAL CONST Robtarget Tr_meulage_motif_1_P149 :=[[123.240265625,-160.491640625,33.13421875],[0.635107748876336,-0.564376918949611,-0.350307497755773,0.394209966502961],[0,0,0,0],[8.999999E+09,8.999999E+09,8.999999E+09,8.999999E+09,8.999999E+09,8.999999E+09]];
	LOCAL CONST Robtarget Tr_meulage_motif_1_P150 :=[[123.7145546875,-159.611265625,33.13420703125],[0.635107748876336,-0.564376918949611,-0.350307497755773,0.394209966502961],[0,0,0,0],[8.999999E+09,8.999999E+09,8.999999E+09,8.999999E+09,8.999999E+09,8.999999E+09]];
	LOCAL CONST Robtarget Tr_meulage_motif_1_P151 :=[[124.1888515625,-158.73090625,33.1341953125],[0.635107748876336,-0.564376918949611,-0.350307497755773,0.394209966502961],[0,0,0,0],[8.999999E+09,8.999999E+09,8.999999E+09,8.999999E+09,8.999999E+09,8.999999E+09]];
	LOCAL CONST Robtarget Tr_meulage_motif_1_P152 :=[[124.663140625,-157.85053125,33.13418359375],[0.635107748876336,-0.564376918949611,-0.350307497755773,0.394209966502961],[0,0,0,0],[8.999999E+09,8.999999E+09,8.999999E+09,8.999999E+09,8.999999E+09,8.999999E+09]];
	LOCAL CONST Robtarget Tr_meulage_motif_1_P153 :=[[125.1374375,-156.970171875,33.13416796875],[0.635107748876336,-0.564376918949611,-0.350307497755773,0.394209966502961],[0,0,0,0],[8.999999E+09,8.999999E+09,8.999999E+09,8.999999E+09,8.999999E+09,8.999999E+09]];
	LOCAL CONST Robtarget Tr_meulage_motif_1_P154 :=[[125.6117265625,-156.089796875,33.13415625],[0.635107748876336,-0.564376918949611,-0.350307497755773,0.394209966502961],[0,0,0,0],[8.999999E+09,8.999999E+09,8.999999E+09,8.999999E+09,8.999999E+09,8.999999E+09]];
	LOCAL CONST Robtarget Tr_meulage_motif_1_P155 :=[[126.0860234375,-155.2094375,33.13414453125],[0.635107748876336,-0.564376918949611,-0.350307497755773,0.394209966502961],[0,0,0,0],[8.999999E+09,8.999999E+09,8.999999E+09,8.999999E+09,8.999999E+09,8.999999E+09]];
	LOCAL CONST Robtarget Tr_meulage_motif_1_P156 :=[[126.5603125,-154.3290625,33.1341328125],[0.635107748876336,-0.564376918949611,-0.350307497755773,0.394209966502961],[0,0,0,0],[8.999999E+09,8.999999E+09,8.999999E+09,8.999999E+09,8.999999E+09,8.999999E+09]];
	LOCAL CONST Robtarget Tr_meulage_motif_1_P157 :=[[127.034609375,-153.448703125,33.13412109375],[0.635107748876336,-0.564376918949611,-0.350307497755773,0.394209966502961],[0,0,0,0],[8.999999E+09,8.999999E+09,8.999999E+09,8.999999E+09,8.999999E+09,8.999999E+09]];
	LOCAL CONST Robtarget Tr_meulage_motif_1_P158 :=[[127.5088984375,-152.568328125,33.134109375],[0.635107748876336,-0.564376918949611,-0.350307497755773,0.394209966502961],[0,0,0,0],[8.999999E+09,8.999999E+09,8.999999E+09,8.999999E+09,8.999999E+09,8.999999E+09]];
	LOCAL CONST Robtarget Tr_meulage_motif_1_P159 :=[[127.98278125,-151.696203125,33.02355859375],[0.635107748876336,-0.564376918949611,-0.350307497755773,0.394209966502961],[0,0,0,0],[8.999999E+09,8.999999E+09,8.999999E+09,8.999999E+09,8.999999E+09,8.999999E+09]];
	LOCAL CONST Robtarget Tr_meulage_motif_1_P160 :=[[128.4376640625,-150.866140625,32.81246875],[0.635107748876336,-0.564376918949611,-0.350307497755773,0.394209966502961],[0,0,0,0],[8.999999E+09,8.999999E+09,8.999999E+09,8.999999E+09,8.999999E+09,8.999999E+09]];
	LOCAL CONST Robtarget Tr_meulage_motif_1_P161 :=[[128.849765625,-150.119578125,32.540751953125],[0.635107748876336,-0.564376918949611,-0.350307497755773,0.394209966502961],[0,0,0,0],[8.999999E+09,8.999999E+09,8.999999E+09,8.999999E+09,8.999999E+09,8.999999E+09]];
	LOCAL CONST Robtarget Tr_meulage_motif_1_P162 :=[[129.2132421875,-149.463546875,32.264947265625],[0.635107748876336,-0.564376918949611,-0.350307497755773,0.394209966502961],[0,0,0,0],[8.999999E+09,8.999999E+09,8.999999E+09,8.999999E+09,8.999999E+09,8.999999E+09]];
	LOCAL CONST Robtarget Tr_meulage_motif_1_P163 :=[[129.7528515625,-148.503578125,31.649125],[0.635107748876336,-0.564376918949611,-0.350307497755773,0.394209966502961],[0,0,0,0],[8.999999E+09,8.999999E+09,8.999999E+09,8.999999E+09,8.999999E+09,8.999999E+09]];
	LOCAL CONST Robtarget Tr_meulage_motif_1_P164 :=[[130.2623828125,-147.61509375,30.801892578125],[0.635107748876336,-0.564376918949611,-0.350307497755773,0.394209966502961],[0,0,0,0],[8.999999E+09,8.999999E+09,8.999999E+09,8.999999E+09,8.999999E+09,8.999999E+09]];
	LOCAL CONST Robtarget Tr_meulage_motif_1_P165 :=[[130.6933046875,-146.884421875,29.778533203125],[0.635107748876336,-0.564376918949611,-0.350307497755773,0.394209966502961],[0,0,0,0],[8.999999E+09,8.999999E+09,8.999999E+09,8.999999E+09,8.999999E+09,8.999999E+09]];
	LOCAL CONST Robtarget Tr_meulage_motif_1_P166 :=[[130.956328125,-146.471640625,28.662912109375],[0.635107748876336,-0.564376918949611,-0.350307497755773,0.394209966502961],[0,0,0,0],[8.999999E+09,8.999999E+09,8.999999E+09,8.999999E+09,8.999999E+09,8.999999E+09]];
	LOCAL CONST Robtarget Tr_meulage_motif_1_P167 :=[[130.988796875,-146.45840625,27.96730078125],[0.635107748876336,-0.564376918949611,-0.350307497755773,0.394209966502961],[0,0,0,0],[8.999999E+09,8.999999E+09,8.999999E+09,8.999999E+09,8.999999E+09,8.999999E+09]];
	LOCAL CONST Robtarget Tr_meulage_motif_1_P168 :=[[131.007453125,-146.46846875,27.306390625],[0.635107748876336,-0.564376918949611,-0.350307497755773,0.394209966502961],[0,0,0,0],[8.999999E+09,8.999999E+09,8.999999E+09,8.999999E+09,8.999999E+09,8.999999E+09]];
	LOCAL CONST Robtarget Tr_meulage_motif_1_P169 :=[[131.000078125,-146.52684375,26.64563671875],[0.635107748876336,-0.564376918949611,-0.350307497755773,0.394209966502961],[0,0,0,0],[8.999999E+09,8.999999E+09,8.999999E+09,8.999999E+09,8.999999E+09,8.999999E+09]];
	LOCAL CONST Robtarget Tr_meulage_motif_1_P170 :=[[130.794859375,-146.98221875,25.544458984375],[0.635107748876336,-0.564376918949611,-0.350307497755773,0.394209966502961],[0,0,0,0],[8.999999E+09,8.999999E+09,8.999999E+09,8.999999E+09,8.999999E+09,8.999999E+09]];
	LOCAL CONST Robtarget Tr_meulage_motif_1_P171 :=[[130.4169609375,-147.751671875,24.53836328125],[0.635107748876336,-0.564376918949611,-0.350307497755773,0.394209966502961],[0,0,0,0],[8.999999E+09,8.999999E+09,8.999999E+09,8.999999E+09,8.999999E+09,8.999999E+09]];
	LOCAL CONST Robtarget Tr_meulage_motif_1_P172 :=[[129.954953125,-148.66525,23.70992578125],[0.635107748876336,-0.564376918949611,-0.350307497755773,0.394209966502961],[0,0,0,0],[8.999999E+09,8.999999E+09,8.999999E+09,8.999999E+09,8.999999E+09,8.999999E+09]];
	LOCAL CONST Robtarget Tr_meulage_motif_1_P173 :=[[129.640234375,-149.276171875,23.314388671875],[0.635107748876336,-0.564376918949611,-0.350307497755773,0.394209966502961],[0,0,0,0],[8.999999E+09,8.999999E+09,8.999999E+09,8.999999E+09,8.999999E+09,8.999999E+09]];
	LOCAL CONST Robtarget Tr_meulage_motif_1_P174 :=[[129.1046875,-150.3031875,22.82712109375],[0.635107748876336,-0.564376918949611,-0.350307497755773,0.394209966502961],[0,0,0,0],[8.999999E+09,8.999999E+09,8.999999E+09,8.999999E+09,8.999999E+09,8.999999E+09]];
	LOCAL CONST Robtarget Tr_meulage_motif_1_P175 :=[[128.71134375,-151.051140625,22.563173828125],[0.635107748876336,-0.564376918949611,-0.350307497755773,0.394209966502961],[0,0,0,0],[8.999999E+09,8.999999E+09,8.999999E+09,8.999999E+09,8.999999E+09,8.999999E+09]];
	LOCAL CONST Robtarget Tr_meulage_motif_1_P176 :=[[128.2750703125,-151.874765625,22.358822265625],[0.635107748876336,-0.564376918949611,-0.350307497755773,0.394209966502961],[0,0,0,0],[8.999999E+09,8.999999E+09,8.999999E+09,8.999999E+09,8.999999E+09,8.999999E+09]];
	LOCAL CONST Robtarget Tr_meulage_motif_1_P177 :=[[127.8125859375,-152.740546875,22.250296875],[0.635107748876336,-0.564376918949611,-0.350307497755773,0.394209966502961],[0,0,0,0],[8.999999E+09,8.999999E+09,8.999999E+09,8.999999E+09,8.999999E+09,8.999999E+09]];
	LOCAL CONST Robtarget Tr_meulage_motif_1_P178 :=[[127.3449453125,-153.616046875,22.139771484375],[0.635107748876336,-0.564376918949611,-0.350307497755773,0.394209966502961],[0,0,0,0],[8.999999E+09,8.999999E+09,8.999999E+09,8.999999E+09,8.999999E+09,8.999999E+09]];
	LOCAL CONST Robtarget Tr_meulage_motif_1_P179 :=[[126.8706484375,-154.496421875,22.13978515625],[0.635107748876336,-0.564376918949611,-0.350307497755773,0.394209966502961],[0,0,0,0],[8.999999E+09,8.999999E+09,8.999999E+09,8.999999E+09,8.999999E+09,8.999999E+09]];
	LOCAL CONST Robtarget Tr_meulage_motif_1_P180 :=[[126.396359375,-155.37678125,22.139796875],[0.635107748876336,-0.564376918949611,-0.350307497755773,0.394209966502961],[0,0,0,0],[8.999999E+09,8.999999E+09,8.999999E+09,8.999999E+09,8.999999E+09,8.999999E+09]];
	LOCAL CONST Robtarget Tr_meulage_motif_1_P181 :=[[125.9220625,-156.25715625,22.13980859375],[0.635107748876336,-0.564376918949611,-0.350307497755773,0.394209966502961],[0,0,0,0],[8.999999E+09,8.999999E+09,8.999999E+09,8.999999E+09,8.999999E+09,8.999999E+09]];
	LOCAL CONST Robtarget Tr_meulage_motif_1_P182 :=[[125.4477734375,-157.137515625,22.139822265625],[0.635107748876336,-0.564376918949611,-0.350307497755773,0.394209966502961],[0,0,0,0],[8.999999E+09,8.999999E+09,8.999999E+09,8.999999E+09,8.999999E+09,8.999999E+09]];
	LOCAL CONST Robtarget Tr_meulage_motif_1_P183 :=[[124.9734765625,-158.017890625,22.139833984375],[0.635107748876336,-0.564376918949611,-0.350307497755773,0.394209966502961],[0,0,0,0],[8.999999E+09,8.999999E+09,8.999999E+09,8.999999E+09,8.999999E+09,8.999999E+09]];
	LOCAL CONST Robtarget Tr_meulage_motif_1_P184 :=[[124.4991875,-158.89825,22.13984765625],[0.635107748876336,-0.564376918949611,-0.350307497755773,0.394209966502961],[0,0,0,0],[8.999999E+09,8.999999E+09,8.999999E+09,8.999999E+09,8.999999E+09,8.999999E+09]];
	LOCAL CONST Robtarget Tr_meulage_motif_1_P185 :=[[124.024890625,-159.778625,22.139859375],[0.635107748876336,-0.564376918949611,-0.350307497755773,0.394209966502961],[0,0,0,0],[8.999999E+09,8.999999E+09,8.999999E+09,8.999999E+09,8.999999E+09,8.999999E+09]];
	LOCAL CONST Robtarget Tr_meulage_motif_1_P186 :=[[123.5506015625,-160.658984375,22.13987109375],[0.635107748876336,-0.564376918949611,-0.350307497755773,0.394209966502961],[0,0,0,0],[8.999999E+09,8.999999E+09,8.999999E+09,8.999999E+09,8.999999E+09,8.999999E+09]];
	LOCAL CONST Robtarget Tr_meulage_motif_1_P187 :=[[123.0763046875,-161.539359375,22.139884765625],[0.635107748876336,-0.564376918949611,-0.350307497755773,0.394209966502961],[0,0,0,0],[8.999999E+09,8.999999E+09,8.999999E+09,8.999999E+09,8.999999E+09,8.999999E+09]];
	LOCAL CONST Robtarget Tr_meulage_motif_1_P188 :=[[122.602015625,-162.41971875,22.139896484375],[0.635107748876336,-0.564376918949611,-0.350307497755773,0.394209966502961],[0,0,0,0],[8.999999E+09,8.999999E+09,8.999999E+09,8.999999E+09,8.999999E+09,8.999999E+09]];
	LOCAL CONST Robtarget Tr_meulage_motif_1_P189 :=[[122.12771875,-163.30009375,22.139908203125],[0.635107748876336,-0.564376918949611,-0.350307497755773,0.394209966502961],[0,0,0,0],[8.999999E+09,8.999999E+09,8.999999E+09,8.999999E+09,8.999999E+09,8.999999E+09]];
	LOCAL CONST Robtarget Tr_meulage_motif_1_P190 :=[[121.6534296875,-164.180453125,22.139921875],[0.635107748876336,-0.564376918949611,-0.350307497755773,0.394209966502961],[0,0,0,0],[8.999999E+09,8.999999E+09,8.999999E+09,8.999999E+09,8.999999E+09,8.999999E+09]];
	LOCAL CONST Robtarget Tr_meulage_motif_1_P191 :=[[121.1791328125,-165.060828125,22.13993359375],[0.635107748876336,-0.564376918949611,-0.350307497755773,0.394209966502961],[0,0,0,0],[8.999999E+09,8.999999E+09,8.999999E+09,8.999999E+09,8.999999E+09,8.999999E+09]];
	LOCAL CONST Robtarget Tr_meulage_motif_1_P192 :=[[120.70484375,-165.9411875,22.139947265625],[0.635107748876336,-0.564376918949611,-0.350307497755773,0.394209966502961],[0,0,0,0],[8.999999E+09,8.999999E+09,8.999999E+09,8.999999E+09,8.999999E+09,8.999999E+09]];
	LOCAL CONST Robtarget Tr_meulage_motif_1_P193 :=[[120.230546875,-166.8215625,22.139958984375],[0.635107748876336,-0.564376918949611,-0.350307497755773,0.394209966502961],[0,0,0,0],[8.999999E+09,8.999999E+09,8.999999E+09,8.999999E+09,8.999999E+09,8.999999E+09]];
	LOCAL CONST Robtarget Tr_meulage_motif_1_P194 :=[[119.7562578125,-167.701921875,22.139970703125],[0.635107748876336,-0.564376918949611,-0.350307497755773,0.394209966502961],[0,0,0,0],[8.999999E+09,8.999999E+09,8.999999E+09,8.999999E+09,8.999999E+09,8.999999E+09]];
	LOCAL CONST Robtarget Tr_meulage_motif_1_P195 :=[[119.2819609375,-168.582296875,22.139984375],[0.635107748876336,-0.564376918949611,-0.350307497755773,0.394209966502961],[0,0,0,0],[8.999999E+09,8.999999E+09,8.999999E+09,8.999999E+09,8.999999E+09,8.999999E+09]];
	LOCAL CONST Robtarget Tr_meulage_motif_1_P196 :=[[118.807671875,-169.46265625,22.13999609375],[0.635107748876336,-0.564376918949611,-0.350307497755773,0.394209966502961],[0,0,0,0],[8.999999E+09,8.999999E+09,8.999999E+09,8.999999E+09,8.999999E+09,8.999999E+09]];
	LOCAL CONST Robtarget Tr_meulage_motif_1_P197 :=[[118.333375,-170.34303125,22.1400078125],[0.635107748876336,-0.564376918949611,-0.350307497755773,0.394209966502961],[0,0,0,0],[8.999999E+09,8.999999E+09,8.999999E+09,8.999999E+09,8.999999E+09,8.999999E+09]];
	LOCAL CONST Robtarget Tr_meulage_motif_1_P198 :=[[117.8590859375,-171.223390625,22.140021484375],[0.635107748876336,-0.564376918949611,-0.350307497755773,0.394209966502961],[0,0,0,0],[8.999999E+09,8.999999E+09,8.999999E+09,8.999999E+09,8.999999E+09,8.999999E+09]];
	LOCAL CONST Robtarget Tr_meulage_motif_1_P199 :=[[117.384796875,-172.103765625,22.140033203125],[0.635107748876336,-0.564376918949611,-0.350307497755773,0.394209966502961],[0,0,0,0],[8.999999E+09,8.999999E+09,8.999999E+09,8.999999E+09,8.999999E+09,8.999999E+09]];
	LOCAL CONST Robtarget Tr_meulage_motif_1_P200 :=[[116.9105,-172.984125,22.140046875],[0.635107748876336,-0.564376918949611,-0.350307497755773,0.394209966502961],[0,0,0,0],[8.999999E+09,8.999999E+09,8.999999E+09,8.999999E+09,8.999999E+09,8.999999E+09]];
	LOCAL CONST Robtarget Tr_meulage_motif_1_P201 :=[[116.4362109375,-173.8645,22.14005859375],[0.635107748876336,-0.564376918949611,-0.350307497755773,0.394209966502961],[0,0,0,0],[8.999999E+09,8.999999E+09,8.999999E+09,8.999999E+09,8.999999E+09,8.999999E+09]];
	LOCAL CONST Robtarget Tr_meulage_motif_1_P202 :=[[115.9619140625,-174.744859375,22.1400703125],[0.635107748876336,-0.564376918949611,-0.350307497755773,0.394209966502961],[0,0,0,0],[8.999999E+09,8.999999E+09,8.999999E+09,8.999999E+09,8.999999E+09,8.999999E+09]];
	LOCAL CONST Robtarget Tr_meulage_motif_1_P203 :=[[115.487625,-175.625234375,22.140083984375],[0.635107748876336,-0.564376918949611,-0.350307497755773,0.394209966502961],[0,0,0,0],[8.999999E+09,8.999999E+09,8.999999E+09,8.999999E+09,8.999999E+09,8.999999E+09]];
	LOCAL CONST Robtarget Tr_meulage_motif_1_P204 :=[[115.013328125,-176.50559375,22.140095703125],[0.635107748876336,-0.564376918949611,-0.350307497755773,0.394209966502961],[0,0,0,0],[8.999999E+09,8.999999E+09,8.999999E+09,8.999999E+09,8.999999E+09,8.999999E+09]];
	LOCAL CONST Robtarget Tr_meulage_motif_1_P205 :=[[114.5390390625,-177.38596875,22.140107421875],[0.635107748876336,-0.564376918949611,-0.350307497755773,0.394209966502961],[0,0,0,0],[8.999999E+09,8.999999E+09,8.999999E+09,8.999999E+09,8.999999E+09,8.999999E+09]];
	LOCAL CONST Robtarget Tr_meulage_motif_1_P206 :=[[114.0647421875,-178.266328125,22.14012109375],[0.635107748876336,-0.564376918949611,-0.350307497755773,0.394209966502961],[0,0,0,0],[8.999999E+09,8.999999E+09,8.999999E+09,8.999999E+09,8.999999E+09,8.999999E+09]];
	LOCAL CONST Robtarget Tr_meulage_motif_1_P207 :=[[113.590453125,-179.146703125,22.1401328125],[0.635107748876336,-0.564376918949611,-0.350307497755773,0.394209966502961],[0,0,0,0],[8.999999E+09,8.999999E+09,8.999999E+09,8.999999E+09,8.999999E+09,8.999999E+09]];
	LOCAL CONST Robtarget Tr_meulage_motif_1_P208 :=[[113.11615625,-180.0270625,22.14014453125],[0.635107748876336,-0.564376918949611,-0.350307497755773,0.394209966502961],[0,0,0,0],[8.999999E+09,8.999999E+09,8.999999E+09,8.999999E+09,8.999999E+09,8.999999E+09]];
	LOCAL CONST Robtarget Tr_meulage_motif_1_P209 :=[[112.6418671875,-180.9074375,22.140158203125],[0.635107748876336,-0.564376918949611,-0.350307497755773,0.394209966502961],[0,0,0,0],[8.999999E+09,8.999999E+09,8.999999E+09,8.999999E+09,8.999999E+09,8.999999E+09]];
	LOCAL CONST Robtarget Tr_meulage_motif_1_P210 :=[[112.1675703125,-181.787796875,22.140169921875],[0.635107748876336,-0.564376918949611,-0.350307497755773,0.394209966502961],[0,0,0,0],[8.999999E+09,8.999999E+09,8.999999E+09,8.999999E+09,8.999999E+09,8.999999E+09]];
	LOCAL CONST Robtarget Tr_meulage_motif_1_P211 :=[[111.69328125,-182.668171875,22.14018359375],[0.635107748876336,-0.564376918949611,-0.350307497755773,0.394209966502961],[0,0,0,0],[8.999999E+09,8.999999E+09,8.999999E+09,8.999999E+09,8.999999E+09,8.999999E+09]];
	LOCAL CONST Robtarget Tr_meulage_motif_1_P212 :=[[111.218984375,-183.54853125,22.1401953125],[0.635107748876336,-0.564376918949611,-0.350307497755773,0.394209966502961],[0,0,0,0],[8.999999E+09,8.999999E+09,8.999999E+09,8.999999E+09,8.999999E+09,8.999999E+09]];
	LOCAL CONST Robtarget Tr_meulage_motif_1_P213 :=[[110.7446953125,-184.42890625,22.14020703125],[0.635107748876336,-0.564376918949611,-0.350307497755773,0.394209966502961],[0,0,0,0],[8.999999E+09,8.999999E+09,8.999999E+09,8.999999E+09,8.999999E+09,8.999999E+09]];
	LOCAL CONST Robtarget Tr_meulage_motif_1_P214 :=[[110.2703984375,-185.309265625,22.140220703125],[0.635107748876336,-0.564376918949611,-0.350307497755773,0.394209966502961],[0,0,0,0],[8.999999E+09,8.999999E+09,8.999999E+09,8.999999E+09,8.999999E+09,8.999999E+09]];
	LOCAL CONST Robtarget Tr_meulage_motif_1_P215 :=[[109.796109375,-186.189640625,22.140232421875],[0.635107748876336,-0.564376918949611,-0.350307497755773,0.394209966502961],[0,0,0,0],[8.999999E+09,8.999999E+09,8.999999E+09,8.999999E+09,8.999999E+09,8.999999E+09]];
	LOCAL CONST Robtarget Tr_meulage_motif_1_P216 :=[[109.3284609375,-187.065140625,22.029708984375],[0.635107748876336,-0.564376918949611,-0.350307497755773,0.394209966502961],[0,0,0,0],[8.999999E+09,8.999999E+09,8.999999E+09,8.999999E+09,8.999999E+09,8.999999E+09]];
	LOCAL CONST Robtarget Tr_meulage_motif_1_P217 :=[[108.8855,-187.901625,21.818640625],[0.635107748876336,-0.564376918949611,-0.350307497755773,0.394209966502961],[0,0,0,0],[8.999999E+09,8.999999E+09,8.999999E+09,8.999999E+09,8.999999E+09,8.999999E+09]];
	LOCAL CONST Robtarget Tr_meulage_motif_1_P218 :=[[108.488734375,-188.656453125,21.546947265625],[0.635107748876336,-0.564376918949611,-0.350307497755773,0.394209966502961],[0,0,0,0],[8.999999E+09,8.999999E+09,8.999999E+09,8.999999E+09,8.999999E+09,8.999999E+09]];
	LOCAL CONST Robtarget Tr_meulage_motif_1_P219 :=[[108.159859375,-189.28746875,21.24297265625],[0.635107748876336,-0.564376918949611,-0.350307497755773,0.394209966502961],[0,0,0,0],[8.999999E+09,8.999999E+09,8.999999E+09,8.999999E+09,8.999999E+09,8.999999E+09]];
	LOCAL CONST Robtarget Tr_meulage_motif_1_P220 :=[[107.68790625,-190.208265625,20.580794921875],[0.635107748876336,-0.564376918949611,-0.350307497755773,0.394209966502961],[0,0,0,0],[8.999999E+09,8.999999E+09,8.999999E+09,8.999999E+09,8.999999E+09,8.999999E+09]];
	LOCAL CONST Robtarget Tr_meulage_motif_1_P221 :=[[107.2855703125,-191.016015625,19.67931640625],[0.635107748876336,-0.564376918949611,-0.350307497755773,0.394209966502961],[0,0,0,0],[8.999999E+09,8.999999E+09,8.999999E+09,8.999999E+09,8.999999E+09,8.999999E+09]];
	LOCAL CONST Robtarget Tr_meulage_motif_1_P222 :=[[107.0613515625,-191.50290625,18.63384375],[0.635107748876336,-0.564376918949611,-0.350307497755773,0.394209966502961],[0,0,0,0],[8.999999E+09,8.999999E+09,8.999999E+09,8.999999E+09,8.999999E+09,8.999999E+09]];
	LOCAL CONST Robtarget Tr_meulage_motif_1_P223 :=[[106.993265625,-191.676125,17.94096875],[0.635107748876336,-0.564376918949611,-0.350307497755773,0.394209966502961],[0,0,0,0],[8.999999E+09,8.999999E+09,8.999999E+09,8.999999E+09,8.999999E+09,8.999999E+09]];
	LOCAL CONST Robtarget Tr_meulage_motif_1_P224 :=[[106.9847109375,-191.744046875,17.171365234375],[0.635107748876336,-0.564376918949611,-0.350307497755773,0.394209966502961],[0,0,0,0],[8.999999E+09,8.999999E+09,8.999999E+09,8.999999E+09,8.999999E+09,8.999999E+09]];
	LOCAL CONST Robtarget Tr_meulage_motif_1_P225 :=[[107.0381796875,-191.696828125,16.401900390625],[0.635107748876336,-0.564376918949611,-0.350307497755773,0.394209966502961],[0,0,0,0],[8.999999E+09,8.999999E+09,8.999999E+09,8.999999E+09,8.999999E+09,8.999999E+09]];
	LOCAL CONST Robtarget Tr_meulage_motif_1_P226 :=[[107.268453125,-191.34428125,15.2942138671875],[0.635107748876336,-0.564376918949611,-0.350307497755773,0.394209966502961],[0,0,0,0],[8.999999E+09,8.999999E+09,8.999999E+09,8.999999E+09,8.999999E+09,8.999999E+09]];
	LOCAL CONST Robtarget Tr_meulage_motif_1_P227 :=[[107.481484375,-190.988453125,14.708822265625],[0.635107748876336,-0.564376918949611,-0.350307497755773,0.394209966502961],[0,0,0,0],[8.999999E+09,8.999999E+09,8.999999E+09,8.999999E+09,8.999999E+09,8.999999E+09]];
	LOCAL CONST Robtarget Tr_meulage_motif_1_P228 :=[[107.927265625,-190.220953125,13.822111328125],[0.635107748876336,-0.564376918949611,-0.350307497755773,0.394209966502961],[0,0,0,0],[8.999999E+09,8.999999E+09,8.999999E+09,8.999999E+09,8.999999E+09,8.999999E+09]];
	LOCAL CONST Robtarget Tr_meulage_motif_1_P229 :=[[108.2167421875,-189.711640625,13.40803515625],[0.635107748876336,-0.564376918949611,-0.350307497755773,0.394209966502961],[0,0,0,0],[8.999999E+09,8.999999E+09,8.999999E+09,8.999999E+09,8.999999E+09,8.999999E+09]];
	LOCAL CONST Robtarget Tr_meulage_motif_1_P230 :=[[108.7623046875,-188.73575,12.86417578125],[0.635107748876336,-0.564376918949611,-0.350307497755773,0.394209966502961],[0,0,0,0],[8.999999E+09,8.999999E+09,8.999999E+09,8.999999E+09,8.999999E+09,8.999999E+09]];
	LOCAL CONST Robtarget Tr_meulage_motif_1_P231 :=[[109.16221875,-188.01340625,12.5688173828125],[0.635107748876336,-0.564376918949611,-0.350307497755773,0.394209966502961],[0,0,0,0],[8.999999E+09,8.999999E+09,8.999999E+09,8.999999E+09,8.999999E+09,8.999999E+09]];
	LOCAL CONST Robtarget Tr_meulage_motif_1_P232 :=[[109.61003125,-187.196015625,12.3644267578125],[0.635107748876336,-0.564376918949611,-0.350307497755773,0.394209966502961],[0,0,0,0],[8.999999E+09,8.999999E+09,8.999999E+09,8.999999E+09,8.999999E+09,8.999999E+09]];
	LOCAL CONST Robtarget Tr_meulage_motif_1_P233 :=[[110.078640625,-186.33353125,12.2559228515625],[0.635107748876336,-0.564376918949611,-0.350307497755773,0.394209966502961],[0,0,0,0],[8.999999E+09,8.999999E+09,8.999999E+09,8.999999E+09,8.999999E+09,8.999999E+09]];
	LOCAL CONST Robtarget Tr_meulage_motif_1_P234 :=[[110.5525234375,-185.46140625,12.1453583984375],[0.635107748876336,-0.564376918949611,-0.350307497755773,0.394209966502961],[0,0,0,0],[8.999999E+09,8.999999E+09,8.999999E+09,8.999999E+09,8.999999E+09,8.999999E+09]];
	LOCAL CONST Robtarget Tr_meulage_motif_1_P235 :=[[111.0268203125,-184.58103125,12.145345703125],[0.635107748876336,-0.564376918949611,-0.350307497755773,0.394209966502961],[0,0,0,0],[8.999999E+09,8.999999E+09,8.999999E+09,8.999999E+09,8.999999E+09,8.999999E+09]];
	LOCAL CONST Robtarget Tr_meulage_motif_1_P236 :=[[111.501109375,-183.700671875,12.1453330078125],[0.635107748876336,-0.564376918949611,-0.350307497755773,0.394209966502961],[0,0,0,0],[8.999999E+09,8.999999E+09,8.999999E+09,8.999999E+09,8.999999E+09,8.999999E+09]];
	LOCAL CONST Robtarget Tr_meulage_motif_1_P237 :=[[111.97540625,-182.820296875,12.1453212890625],[0.635107748876336,-0.564376918949611,-0.350307497755773,0.394209966502961],[0,0,0,0],[8.999999E+09,8.999999E+09,8.999999E+09,8.999999E+09,8.999999E+09,8.999999E+09]];
	LOCAL CONST Robtarget Tr_meulage_motif_1_P238 :=[[112.4496953125,-181.9399375,12.14530859375],[0.635107748876336,-0.564376918949611,-0.350307497755773,0.394209966502961],[0,0,0,0],[8.999999E+09,8.999999E+09,8.999999E+09,8.999999E+09,8.999999E+09,8.999999E+09]];
	LOCAL CONST Robtarget Tr_meulage_motif_1_P239 :=[[112.923984375,-181.0595625,12.1452958984375],[0.635107748876336,-0.564376918949611,-0.350307497755773,0.394209966502961],[0,0,0,0],[8.999999E+09,8.999999E+09,8.999999E+09,8.999999E+09,8.999999E+09,8.999999E+09]];
	LOCAL CONST Robtarget Tr_meulage_motif_1_P240 :=[[113.39828125,-180.179203125,12.1452841796875],[0.635107748876336,-0.564376918949611,-0.350307497755773,0.394209966502961],[0,0,0,0],[8.999999E+09,8.999999E+09,8.999999E+09,8.999999E+09,8.999999E+09,8.999999E+09]];
	LOCAL CONST Robtarget Tr_meulage_motif_1_P241 :=[[113.8725703125,-179.298828125,12.145271484375],[0.635107748876336,-0.564376918949611,-0.350307497755773,0.394209966502961],[0,0,0,0],[8.999999E+09,8.999999E+09,8.999999E+09,8.999999E+09,8.999999E+09,8.999999E+09]];
	LOCAL CONST Robtarget Tr_meulage_motif_1_P242 :=[[114.3468671875,-178.41846875,12.1452587890625],[0.635107748876336,-0.564376918949611,-0.350307497755773,0.394209966502961],[0,0,0,0],[8.999999E+09,8.999999E+09,8.999999E+09,8.999999E+09,8.999999E+09,8.999999E+09]];
	LOCAL CONST Robtarget Tr_meulage_motif_1_P243 :=[[114.82115625,-177.53809375,12.14524609375],[0.635107748876336,-0.564376918949611,-0.350307497755773,0.394209966502961],[0,0,0,0],[8.999999E+09,8.999999E+09,8.999999E+09,8.999999E+09,8.999999E+09,8.999999E+09]];
	LOCAL CONST Robtarget Tr_meulage_motif_1_P244 :=[[115.295453125,-176.657734375,12.145234375],[0.635107748876336,-0.564376918949611,-0.350307497755773,0.394209966502961],[0,0,0,0],[8.999999E+09,8.999999E+09,8.999999E+09,8.999999E+09,8.999999E+09,8.999999E+09]];
	LOCAL CONST Robtarget Tr_meulage_motif_1_P245 :=[[115.7697421875,-175.777359375,12.1452216796875],[0.635107748876336,-0.564376918949611,-0.350307497755773,0.394209966502961],[0,0,0,0],[8.999999E+09,8.999999E+09,8.999999E+09,8.999999E+09,8.999999E+09,8.999999E+09]];
	LOCAL CONST Robtarget Tr_meulage_motif_1_P246 :=[[116.2440390625,-174.897,12.145208984375],[0.635107748876336,-0.564376918949611,-0.350307497755773,0.394209966502961],[0,0,0,0],[8.999999E+09,8.999999E+09,8.999999E+09,8.999999E+09,8.999999E+09,8.999999E+09]];
	LOCAL CONST Robtarget Tr_meulage_motif_1_P247 :=[[116.718328125,-174.016625,12.1451962890625],[0.635107748876336,-0.564376918949611,-0.350307497755773,0.394209966502961],[0,0,0,0],[8.999999E+09,8.999999E+09,8.999999E+09,8.999999E+09,8.999999E+09,8.999999E+09]];
	LOCAL CONST Robtarget Tr_meulage_motif_1_P248 :=[[117.192625,-173.136265625,12.1451845703125],[0.635107748876336,-0.564376918949611,-0.350307497755773,0.394209966502961],[0,0,0,0],[8.999999E+09,8.999999E+09,8.999999E+09,8.999999E+09,8.999999E+09,8.999999E+09]];
	LOCAL CONST Robtarget Tr_meulage_motif_1_P249 :=[[117.6669140625,-172.255890625,12.145171875],[0.635107748876336,-0.564376918949611,-0.350307497755773,0.394209966502961],[0,0,0,0],[8.999999E+09,8.999999E+09,8.999999E+09,8.999999E+09,8.999999E+09,8.999999E+09]];
	LOCAL CONST Robtarget Tr_meulage_motif_1_P250 :=[[118.1412109375,-171.37553125,12.1451591796875],[0.635107748876336,-0.564376918949611,-0.350307497755773,0.394209966502961],[0,0,0,0],[8.999999E+09,8.999999E+09,8.999999E+09,8.999999E+09,8.999999E+09,8.999999E+09]];
	LOCAL CONST Robtarget Tr_meulage_motif_1_P251 :=[[118.6155,-170.49515625,12.145146484375],[0.635107748876336,-0.564376918949611,-0.350307497755773,0.394209966502961],[0,0,0,0],[8.999999E+09,8.999999E+09,8.999999E+09,8.999999E+09,8.999999E+09,8.999999E+09]];
	LOCAL CONST Robtarget Tr_meulage_motif_1_P252 :=[[119.089796875,-169.614796875,12.145134765625],[0.635107748876336,-0.564376918949611,-0.350307497755773,0.394209966502961],[0,0,0,0],[8.999999E+09,8.999999E+09,8.999999E+09,8.999999E+09,8.999999E+09,8.999999E+09]];
	LOCAL CONST Robtarget Tr_meulage_motif_1_P253 :=[[119.5640859375,-168.734421875,12.1451220703125],[0.635107748876336,-0.564376918949611,-0.350307497755773,0.394209966502961],[0,0,0,0],[8.999999E+09,8.999999E+09,8.999999E+09,8.999999E+09,8.999999E+09,8.999999E+09]];
	LOCAL CONST Robtarget Tr_meulage_motif_1_P254 :=[[120.0383828125,-167.8540625,12.145109375],[0.635107748876336,-0.564376918949611,-0.350307497755773,0.394209966502961],[0,0,0,0],[8.999999E+09,8.999999E+09,8.999999E+09,8.999999E+09,8.999999E+09,8.999999E+09]];
	LOCAL CONST Robtarget Tr_meulage_motif_1_P255 :=[[120.512671875,-166.9736875,12.1450966796875],[0.635107748876336,-0.564376918949611,-0.350307497755773,0.394209966502961],[0,0,0,0],[8.999999E+09,8.999999E+09,8.999999E+09,8.999999E+09,8.999999E+09,8.999999E+09]];
	LOCAL CONST Robtarget Tr_meulage_motif_1_P256 :=[[120.98696875,-166.093328125,12.1450849609375],[0.635107748876336,-0.564376918949611,-0.350307497755773,0.394209966502961],[0,0,0,0],[8.999999E+09,8.999999E+09,8.999999E+09,8.999999E+09,8.999999E+09,8.999999E+09]];
	LOCAL CONST Robtarget Tr_meulage_motif_1_P257 :=[[121.4612578125,-165.212953125,12.145072265625],[0.635107748876336,-0.564376918949611,-0.350307497755773,0.394209966502961],[0,0,0,0],[8.999999E+09,8.999999E+09,8.999999E+09,8.999999E+09,8.999999E+09,8.999999E+09]];
	LOCAL CONST Robtarget Tr_meulage_motif_1_P258 :=[[121.9355546875,-164.33259375,12.1450595703125],[0.635107748876336,-0.564376918949611,-0.350307497755773,0.394209966502961],[0,0,0,0],[8.999999E+09,8.999999E+09,8.999999E+09,8.999999E+09,8.999999E+09,8.999999E+09]];
	LOCAL CONST Robtarget Tr_meulage_motif_1_P259 :=[[122.40984375,-163.45221875,12.145046875],[0.635107748876336,-0.564376918949611,-0.350307497755773,0.394209966502961],[0,0,0,0],[8.999999E+09,8.999999E+09,8.999999E+09,8.999999E+09,8.999999E+09,8.999999E+09]];
	LOCAL CONST Robtarget Tr_meulage_motif_1_P260 :=[[122.8841328125,-162.571859375,12.14503515625],[0.635107748876336,-0.564376918949611,-0.350307497755773,0.394209966502961],[0,0,0,0],[8.999999E+09,8.999999E+09,8.999999E+09,8.999999E+09,8.999999E+09,8.999999E+09]];
	LOCAL CONST Robtarget Tr_meulage_motif_1_P261 :=[[123.3584296875,-161.691484375,12.1450224609375],[0.635107748876336,-0.564376918949611,-0.350307497755773,0.394209966502961],[0,0,0,0],[8.999999E+09,8.999999E+09,8.999999E+09,8.999999E+09,8.999999E+09,8.999999E+09]];
	LOCAL CONST Robtarget Tr_meulage_motif_1_P262 :=[[123.83271875,-160.811125,12.145009765625],[0.635107748876336,-0.564376918949611,-0.350307497755773,0.394209966502961],[0,0,0,0],[8.999999E+09,8.999999E+09,8.999999E+09,8.999999E+09,8.999999E+09,8.999999E+09]];
	LOCAL CONST Robtarget Tr_meulage_motif_1_P263 :=[[124.307015625,-159.93075,12.1449970703125],[0.635107748876336,-0.564376918949611,-0.350307497755773,0.394209966502961],[0,0,0,0],[8.999999E+09,8.999999E+09,8.999999E+09,8.999999E+09,8.999999E+09,8.999999E+09]];
	LOCAL CONST Robtarget Tr_meulage_motif_1_P264 :=[[124.7813046875,-159.050390625,12.1449853515625],[0.635107748876336,-0.564376918949611,-0.350307497755773,0.394209966502961],[0,0,0,0],[8.999999E+09,8.999999E+09,8.999999E+09,8.999999E+09,8.999999E+09,8.999999E+09]];
	LOCAL CONST Robtarget Tr_meulage_motif_1_P265 :=[[125.2556015625,-158.170015625,12.14497265625],[0.635107748876336,-0.564376918949611,-0.350307497755773,0.394209966502961],[0,0,0,0],[8.999999E+09,8.999999E+09,8.999999E+09,8.999999E+09,8.999999E+09,8.999999E+09]];
	LOCAL CONST Robtarget Tr_meulage_motif_1_P266 :=[[125.729890625,-157.28965625,12.1449599609375],[0.635107748876336,-0.564376918949611,-0.350307497755773,0.394209966502961],[0,0,0,0],[8.999999E+09,8.999999E+09,8.999999E+09,8.999999E+09,8.999999E+09,8.999999E+09]];
	LOCAL CONST Robtarget Tr_meulage_motif_1_P267 :=[[126.2041875,-156.40928125,12.144947265625],[0.635107748876336,-0.564376918949611,-0.350307497755773,0.394209966502961],[0,0,0,0],[8.999999E+09,8.999999E+09,8.999999E+09,8.999999E+09,8.999999E+09,8.999999E+09]];
	LOCAL CONST Robtarget Tr_meulage_motif_1_P268 :=[[126.6784765625,-155.528921875,12.144935546875],[0.635107748876336,-0.564376918949611,-0.350307497755773,0.394209966502961],[0,0,0,0],[8.999999E+09,8.999999E+09,8.999999E+09,8.999999E+09,8.999999E+09,8.999999E+09]];
	LOCAL CONST Robtarget Tr_meulage_motif_1_P269 :=[[127.1527734375,-154.648546875,12.1449228515625],[0.635107748876336,-0.564376918949611,-0.350307497755773,0.394209966502961],[0,0,0,0],[8.999999E+09,8.999999E+09,8.999999E+09,8.999999E+09,8.999999E+09,8.999999E+09]];
	LOCAL CONST Robtarget Tr_meulage_motif_1_P270 :=[[127.6270625,-153.7681875,12.14491015625],[0.635107748876336,-0.564376918949611,-0.350307497755773,0.394209966502961],[0,0,0,0],[8.999999E+09,8.999999E+09,8.999999E+09,8.999999E+09,8.999999E+09,8.999999E+09]];
	LOCAL CONST Robtarget Tr_meulage_motif_1_P271 :=[[128.101359375,-152.8878125,12.1448974609375],[0.635107748876336,-0.564376918949611,-0.350307497755773,0.394209966502961],[0,0,0,0],[8.999999E+09,8.999999E+09,8.999999E+09,8.999999E+09,8.999999E+09,8.999999E+09]];
	LOCAL CONST Robtarget Tr_meulage_motif_1_P272 :=[[128.5752421875,-152.015671875,12.0343330078125],[0.635107748876336,-0.564376918949611,-0.350307497755773,0.394209966502961],[0,0,0,0],[8.999999E+09,8.999999E+09,8.999999E+09,8.999999E+09,8.999999E+09,8.999999E+09]];
	LOCAL CONST Robtarget Tr_meulage_motif_1_P273 :=[[129.0301171875,-151.185625,11.8232421875],[0.635107748876336,-0.564376918949611,-0.350307497755773,0.394209966502961],[0,0,0,0],[8.999999E+09,8.999999E+09,8.999999E+09,8.999999E+09,8.999999E+09,8.999999E+09]];
	LOCAL CONST Robtarget Tr_meulage_motif_1_P274 :=[[129.4422265625,-150.439046875,11.55154296875],[0.635107748876336,-0.564376918949611,-0.350307497755773,0.394209966502961],[0,0,0,0],[8.999999E+09,8.999999E+09,8.999999E+09,8.999999E+09,8.999999E+09,8.999999E+09]];
	LOCAL CONST Robtarget Tr_meulage_motif_1_P275 :=[[129.805703125,-149.78303125,11.27573828125],[0.635107748876336,-0.564376918949611,-0.350307497755773,0.394209966502961],[0,0,0,0],[8.999999E+09,8.999999E+09,8.999999E+09,8.999999E+09,8.999999E+09,8.999999E+09]];
	LOCAL CONST Robtarget Tr_meulage_motif_1_P276 :=[[130.3453125,-148.8230625,10.659916015625],[0.635107748876336,-0.564376918949611,-0.350307497755773,0.394209966502961],[0,0,0,0],[8.999999E+09,8.999999E+09,8.999999E+09,8.999999E+09,8.999999E+09,8.999999E+09]];
	LOCAL CONST Robtarget Tr_meulage_motif_1_P277 :=[[130.85484375,-147.934578125,9.8126982421875],[0.635107748876336,-0.564376918949611,-0.350307497755773,0.394209966502961],[0,0,0,0],[8.999999E+09,8.999999E+09,8.999999E+09,8.999999E+09,8.999999E+09,8.999999E+09]];
	LOCAL CONST Robtarget Tr_meulage_motif_1_P278 :=[[131.285765625,-147.20390625,8.7893544921875],[0.635107748876336,-0.564376918949611,-0.350307497755773,0.394209966502961],[0,0,0,0],[8.999999E+09,8.999999E+09,8.999999E+09,8.999999E+09,8.999999E+09,8.999999E+09]];
	LOCAL CONST Robtarget Tr_meulage_motif_1_P279 :=[[131.54878125,-146.791125,7.6736875],[0.635107748876336,-0.564376918949611,-0.350307497755773,0.394209966502961],[0,0,0,0],[8.999999E+09,8.999999E+09,8.999999E+09,8.999999E+09,8.999999E+09,8.999999E+09]];
	LOCAL CONST Robtarget Tr_meulage_motif_1_P280 :=[[131.58125,-146.777890625,6.97810693359375],[0.635107748876336,-0.564376918949611,-0.350307497755773,0.394209966502961],[0,0,0,0],[8.999999E+09,8.999999E+09,8.999999E+09,8.999999E+09,8.999999E+09,8.999999E+09]];
	LOCAL CONST Robtarget Tr_meulage_motif_1_P281 :=[[131.59990625,-146.787953125,6.31716552734375],[0.635107748876336,-0.564376918949611,-0.350307497755773,0.394209966502961],[0,0,0,0],[8.999999E+09,8.999999E+09,8.999999E+09,8.999999E+09,8.999999E+09,8.999999E+09]];
	LOCAL CONST Robtarget Tr_meulage_motif_1_P282 :=[[131.59253125,-146.8463125,5.656427734375],[0.635107748876336,-0.564376918949611,-0.350307497755773,0.394209966502961],[0,0,0,0],[8.999999E+09,8.999999E+09,8.999999E+09,8.999999E+09,8.999999E+09,8.999999E+09]];
	LOCAL CONST Robtarget Tr_meulage_motif_1_P283 :=[[131.3873125,-147.3016875,4.555265625],[0.635107748876336,-0.564376918949611,-0.350307497755773,0.394209966502961],[0,0,0,0],[8.999999E+09,8.999999E+09,8.999999E+09,8.999999E+09,8.999999E+09,8.999999E+09]];
	LOCAL CONST Robtarget Tr_meulage_motif_1_P284 :=[[131.009421875,-148.07115625,3.54915307617188],[0.635107748876336,-0.564376918949611,-0.350307497755773,0.394209966502961],[0,0,0,0],[8.999999E+09,8.999999E+09,8.999999E+09,8.999999E+09,8.999999E+09,8.999999E+09]];
	LOCAL CONST Robtarget Tr_meulage_motif_1_P285 :=[[130.5474140625,-148.984734375,2.72073217773438],[0.635107748876336,-0.564376918949611,-0.350307497755773,0.394209966502961],[0,0,0,0],[8.999999E+09,8.999999E+09,8.999999E+09,8.999999E+09,8.999999E+09,8.999999E+09]];
	LOCAL CONST Robtarget Tr_meulage_motif_1_P286 :=[[130.2326953125,-149.59565625,2.32517846679688],[0.635107748876336,-0.564376918949611,-0.350307497755773,0.394209966502961],[0,0,0,0],[8.999999E+09,8.999999E+09,8.999999E+09,8.999999E+09,8.999999E+09,8.999999E+09]];
	LOCAL CONST Robtarget Tr_meulage_motif_1_P287 :=[[129.697140625,-150.622671875,1.83791223144531],[0.635107748876336,-0.564376918949611,-0.350307497755773,0.394209966502961],[0,0,0,0],[8.999999E+09,8.999999E+09,8.999999E+09,8.999999E+09,8.999999E+09,8.999999E+09]];
	LOCAL CONST Robtarget Tr_meulage_motif_1_P288 :=[[129.3038046875,-151.370625,1.57394909667969],[0.635107748876336,-0.564376918949611,-0.350307497755773,0.394209966502961],[0,0,0,0],[8.999999E+09,8.999999E+09,8.999999E+09,8.999999E+09,8.999999E+09,8.999999E+09]];
	LOCAL CONST Robtarget Tr_meulage_motif_1_P289 :=[[128.86753125,-152.194234375,1.36958142089844],[0.635107748876336,-0.564376918949611,-0.350307497755773,0.394209966502961],[0,0,0,0],[8.999999E+09,8.999999E+09,8.999999E+09,8.999999E+09,8.999999E+09,8.999999E+09]];
	LOCAL CONST Robtarget Tr_meulage_motif_1_P290 :=[[128.405046875,-153.06003125,1.2611025390625],[0.635107748876336,-0.564376918949611,-0.350307497755773,0.394209966502961],[0,0,0,0],[8.999999E+09,8.999999E+09,8.999999E+09,8.999999E+09,8.999999E+09,8.999999E+09]];
	LOCAL CONST Robtarget Tr_meulage_motif_1_P291 :=[[127.9373984375,-153.93553125,1.15056225585938],[0.635107748876336,-0.564376918949611,-0.350307497755773,0.394209966502961],[0,0,0,0],[8.999999E+09,8.999999E+09,8.999999E+09,8.999999E+09,8.999999E+09,8.999999E+09]];
	LOCAL CONST Robtarget Tr_meulage_motif_1_P292 :=[[127.463109375,-154.815890625,1.15057470703125],[0.635107748876336,-0.564376918949611,-0.350307497755773,0.394209966502961],[0,0,0,0],[8.999999E+09,8.999999E+09,8.999999E+09,8.999999E+09,8.999999E+09,8.999999E+09]];
	LOCAL CONST Robtarget Tr_meulage_motif_1_P293 :=[[126.9888125,-155.696265625,1.15058715820313],[0.635107748876336,-0.564376918949611,-0.350307497755773,0.394209966502961],[0,0,0,0],[8.999999E+09,8.999999E+09,8.999999E+09,8.999999E+09,8.999999E+09,8.999999E+09]];
	LOCAL CONST Robtarget Tr_meulage_motif_1_P294 :=[[126.5145234375,-156.576625,1.150599609375],[0.635107748876336,-0.564376918949611,-0.350307497755773,0.394209966502961],[0,0,0,0],[8.999999E+09,8.999999E+09,8.999999E+09,8.999999E+09,8.999999E+09,8.999999E+09]];
	LOCAL CONST Robtarget Tr_meulage_motif_1_P295 :=[[126.0402265625,-157.457,1.15061206054688],[0.635107748876336,-0.564376918949611,-0.350307497755773,0.394209966502961],[0,0,0,0],[8.999999E+09,8.999999E+09,8.999999E+09,8.999999E+09,8.999999E+09,8.999999E+09]];
	LOCAL CONST Robtarget Tr_meulage_motif_1_P296 :=[[125.5659375,-158.337359375,1.15062451171875],[0.635107748876336,-0.564376918949611,-0.350307497755773,0.394209966502961],[0,0,0,0],[8.999999E+09,8.999999E+09,8.999999E+09,8.999999E+09,8.999999E+09,8.999999E+09]];
	LOCAL CONST Robtarget Tr_meulage_motif_1_P297 :=[[125.091640625,-159.217734375,1.15063696289063],[0.635107748876336,-0.564376918949611,-0.350307497755773,0.394209966502961],[0,0,0,0],[8.999999E+09,8.999999E+09,8.999999E+09,8.999999E+09,8.999999E+09,8.999999E+09]];
	LOCAL CONST Robtarget Tr_meulage_motif_1_P298 :=[[124.6173515625,-160.09809375,1.1506494140625],[0.635107748876336,-0.564376918949611,-0.350307497755773,0.394209966502961],[0,0,0,0],[8.999999E+09,8.999999E+09,8.999999E+09,8.999999E+09,8.999999E+09,8.999999E+09]];
	LOCAL CONST Robtarget Tr_meulage_motif_1_P299 :=[[124.1430546875,-160.97846875,1.15066186523437],[0.635107748876336,-0.564376918949611,-0.350307497755773,0.394209966502961],[0,0,0,0],[8.999999E+09,8.999999E+09,8.999999E+09,8.999999E+09,8.999999E+09,8.999999E+09]];
	LOCAL CONST Robtarget Tr_meulage_motif_1_P300 :=[[123.668765625,-161.858828125,1.15067431640625],[0.635107748876336,-0.564376918949611,-0.350307497755773,0.394209966502961],[0,0,0,0],[8.999999E+09,8.999999E+09,8.999999E+09,8.999999E+09,8.999999E+09,8.999999E+09]];
	LOCAL CONST Robtarget Tr_meulage_motif_1_P301 :=[[123.19446875,-162.739203125,1.15068676757812],[0.635107748876336,-0.564376918949611,-0.350307497755773,0.394209966502961],[0,0,0,0],[8.999999E+09,8.999999E+09,8.999999E+09,8.999999E+09,8.999999E+09,8.999999E+09]];
	LOCAL CONST Robtarget Tr_meulage_motif_1_P302 :=[[122.7201796875,-163.6195625,1.15069921875],[0.635107748876336,-0.564376918949611,-0.350307497755773,0.394209966502961],[0,0,0,0],[8.999999E+09,8.999999E+09,8.999999E+09,8.999999E+09,8.999999E+09,8.999999E+09]];
	LOCAL CONST Robtarget Tr_meulage_motif_1_P303 :=[[122.2458828125,-164.4999375,1.15071166992188],[0.635107748876336,-0.564376918949611,-0.350307497755773,0.394209966502961],[0,0,0,0],[8.999999E+09,8.999999E+09,8.999999E+09,8.999999E+09,8.999999E+09,8.999999E+09]];
	LOCAL CONST Robtarget Tr_meulage_motif_1_P304 :=[[121.77159375,-165.380296875,1.15072412109375],[0.635107748876336,-0.564376918949611,-0.350307497755773,0.394209966502961],[0,0,0,0],[8.999999E+09,8.999999E+09,8.999999E+09,8.999999E+09,8.999999E+09,8.999999E+09]];
	LOCAL CONST Robtarget Tr_meulage_motif_1_P305 :=[[121.297296875,-166.260671875,1.15073657226563],[0.635107748876336,-0.564376918949611,-0.350307497755773,0.394209966502961],[0,0,0,0],[8.999999E+09,8.999999E+09,8.999999E+09,8.999999E+09,8.999999E+09,8.999999E+09]];
	LOCAL CONST Robtarget Tr_meulage_motif_1_P306 :=[[120.8230078125,-167.14103125,1.1507490234375],[0.635107748876336,-0.564376918949611,-0.350307497755773,0.394209966502961],[0,0,0,0],[8.999999E+09,8.999999E+09,8.999999E+09,8.999999E+09,8.999999E+09,8.999999E+09]];
	LOCAL CONST Robtarget Tr_meulage_motif_1_P307 :=[[120.34871875,-168.02140625,1.15076147460938],[0.635107748876336,-0.564376918949611,-0.350307497755773,0.394209966502961],[0,0,0,0],[8.999999E+09,8.999999E+09,8.999999E+09,8.999999E+09,8.999999E+09,8.999999E+09]];
	LOCAL CONST Robtarget Tr_meulage_motif_1_P308 :=[[119.874421875,-168.901765625,1.15077392578125],[0.635107748876336,-0.564376918949611,-0.350307497755773,0.394209966502961],[0,0,0,0],[8.999999E+09,8.999999E+09,8.999999E+09,8.999999E+09,8.999999E+09,8.999999E+09]];
	LOCAL CONST Robtarget Tr_meulage_motif_1_P309 :=[[119.4001328125,-169.782140625,1.15078637695313],[0.635107748876336,-0.564376918949611,-0.350307497755773,0.394209966502961],[0,0,0,0],[8.999999E+09,8.999999E+09,8.999999E+09,8.999999E+09,8.999999E+09,8.999999E+09]];
	LOCAL CONST Robtarget Tr_meulage_motif_1_P310 :=[[118.9258359375,-170.6625,1.150798828125],[0.635107748876336,-0.564376918949611,-0.350307497755773,0.394209966502961],[0,0,0,0],[8.999999E+09,8.999999E+09,8.999999E+09,8.999999E+09,8.999999E+09,8.999999E+09]];
	LOCAL CONST Robtarget Tr_meulage_motif_1_P311 :=[[118.451546875,-171.542875,1.15081127929687],[0.635107748876336,-0.564376918949611,-0.350307497755773,0.394209966502961],[0,0,0,0],[8.999999E+09,8.999999E+09,8.999999E+09,8.999999E+09,8.999999E+09,8.999999E+09]];
	LOCAL CONST Robtarget Tr_meulage_motif_1_P312 :=[[117.97725,-172.423234375,1.15082373046875],[0.635107748876336,-0.564376918949611,-0.350307497755773,0.394209966502961],[0,0,0,0],[8.999999E+09,8.999999E+09,8.999999E+09,8.999999E+09,8.999999E+09,8.999999E+09]];
	LOCAL CONST Robtarget Tr_meulage_motif_1_P313 :=[[117.5029609375,-173.303609375,1.15083618164062],[0.635107748876336,-0.564376918949611,-0.350307497755773,0.394209966502961],[0,0,0,0],[8.999999E+09,8.999999E+09,8.999999E+09,8.999999E+09,8.999999E+09,8.999999E+09]];
	LOCAL CONST Robtarget Tr_meulage_motif_1_P314 :=[[117.0286640625,-174.18396875,1.1508486328125],[0.635107748876336,-0.564376918949611,-0.350307497755773,0.394209966502961],[0,0,0,0],[8.999999E+09,8.999999E+09,8.999999E+09,8.999999E+09,8.999999E+09,8.999999E+09]];
	LOCAL CONST Robtarget Tr_meulage_motif_1_P315 :=[[116.554375,-175.06434375,1.15086108398437],[0.635107748876336,-0.564376918949611,-0.350307497755773,0.394209966502961],[0,0,0,0],[8.999999E+09,8.999999E+09,8.999999E+09,8.999999E+09,8.999999E+09,8.999999E+09]];
	LOCAL CONST Robtarget Tr_meulage_motif_1_P316 :=[[116.080078125,-175.944703125,1.15087353515625],[0.635107748876336,-0.564376918949611,-0.350307497755773,0.394209966502961],[0,0,0,0],[8.999999E+09,8.999999E+09,8.999999E+09,8.999999E+09,8.999999E+09,8.999999E+09]];
	LOCAL CONST Robtarget Tr_meulage_motif_1_P317 :=[[115.6057890625,-176.825078125,1.15088598632813],[0.635107748876336,-0.564376918949611,-0.350307497755773,0.394209966502961],[0,0,0,0],[8.999999E+09,8.999999E+09,8.999999E+09,8.999999E+09,8.999999E+09,8.999999E+09]];
	LOCAL CONST Robtarget Tr_meulage_motif_1_P318 :=[[115.1314921875,-177.7054375,1.1508984375],[0.635107748876336,-0.564376918949611,-0.350307497755773,0.394209966502961],[0,0,0,0],[8.999999E+09,8.999999E+09,8.999999E+09,8.999999E+09,8.999999E+09,8.999999E+09]];
	LOCAL CONST Robtarget Tr_meulage_motif_1_P319 :=[[114.657203125,-178.5858125,1.15091088867188],[0.635107748876336,-0.564376918949611,-0.350307497755773,0.394209966502961],[0,0,0,0],[8.999999E+09,8.999999E+09,8.999999E+09,8.999999E+09,8.999999E+09,8.999999E+09]];
	LOCAL CONST Robtarget Tr_meulage_motif_1_P320 :=[[114.18290625,-179.466171875,1.15092333984375],[0.635107748876336,-0.564376918949611,-0.350307497755773,0.394209966502961],[0,0,0,0],[8.999999E+09,8.999999E+09,8.999999E+09,8.999999E+09,8.999999E+09,8.999999E+09]];
	LOCAL CONST Robtarget Tr_meulage_motif_1_P321 :=[[113.7086171875,-180.346546875,1.15093579101563],[0.635107748876336,-0.564376918949611,-0.350307497755773,0.394209966502961],[0,0,0,0],[8.999999E+09,8.999999E+09,8.999999E+09,8.999999E+09,8.999999E+09,8.999999E+09]];
	LOCAL CONST Robtarget Tr_meulage_motif_1_P322 :=[[113.2343203125,-181.22690625,1.15094812011719],[0.635107748876336,-0.564376918949611,-0.350307497755773,0.394209966502961],[0,0,0,0],[8.999999E+09,8.999999E+09,8.999999E+09,8.999999E+09,8.999999E+09,8.999999E+09]];
	LOCAL CONST Robtarget Tr_meulage_motif_1_P323 :=[[112.76003125,-182.10728125,1.15096057128906],[0.635107748876336,-0.564376918949611,-0.350307497755773,0.394209966502961],[0,0,0,0],[8.999999E+09,8.999999E+09,8.999999E+09,8.999999E+09,8.999999E+09,8.999999E+09]];
	LOCAL CONST Robtarget Tr_meulage_motif_1_P324 :=[[112.285734375,-182.987640625,1.15097302246094],[0.635107748876336,-0.564376918949611,-0.350307497755773,0.394209966502961],[0,0,0,0],[8.999999E+09,8.999999E+09,8.999999E+09,8.999999E+09,8.999999E+09,8.999999E+09]];
	LOCAL CONST Robtarget Tr_meulage_motif_1_P325 :=[[111.8114453125,-183.868015625,1.15098547363281],[0.635107748876336,-0.564376918949611,-0.350307497755773,0.394209966502961],[0,0,0,0],[8.999999E+09,8.999999E+09,8.999999E+09,8.999999E+09,8.999999E+09,8.999999E+09]];
	LOCAL CONST Robtarget Tr_meulage_motif_1_P326 :=[[111.3371484375,-184.748375,1.15099792480469],[0.635107748876336,-0.564376918949611,-0.350307497755773,0.394209966502961],[0,0,0,0],[8.999999E+09,8.999999E+09,8.999999E+09,8.999999E+09,8.999999E+09,8.999999E+09]];
	LOCAL CONST Robtarget Tr_meulage_motif_1_P327 :=[[110.862859375,-185.62875,1.15101037597656],[0.635107748876336,-0.564376918949611,-0.350307497755773,0.394209966502961],[0,0,0,0],[8.999999E+09,8.999999E+09,8.999999E+09,8.999999E+09,8.999999E+09,8.999999E+09]];
	LOCAL CONST Robtarget Tr_meulage_motif_1_P328 :=[[110.3885703125,-186.509109375,1.15102282714844],[0.635107748876336,-0.564376918949611,-0.350307497755773,0.394209966502961],[0,0,0,0],[8.999999E+09,8.999999E+09,8.999999E+09,8.999999E+09,8.999999E+09,8.999999E+09]];
	LOCAL CONST Robtarget Tr_meulage_motif_1_P329 :=[[109.9142734375,-187.389484375,1.15103527832031],[0.635107748876336,-0.564376918949611,-0.350307497755773,0.394209966502961],[0,0,0,0],[8.999999E+09,8.999999E+09,8.999999E+09,8.999999E+09,8.999999E+09,8.999999E+09]];
	LOCAL CONST Robtarget Tr_meulage_motif_1_P330 :=[[109.439984375,-188.26984375,1.15104772949219],[0.635107748876336,-0.564376918949611,-0.350307497755773,0.394209966502961],[0,0,0,0],[8.999999E+09,8.999999E+09,8.999999E+09,8.999999E+09,8.999999E+09,8.999999E+09]];
	LOCAL CONST Robtarget Tr_meulage_motif_1_P331 :=[[108.9656875,-189.15021875,1.15106018066406],[0.635107748876336,-0.564376918949611,-0.350307497755773,0.394209966502961],[0,0,0,0],[8.999999E+09,8.999999E+09,8.999999E+09,8.999999E+09,8.999999E+09,8.999999E+09]];
	LOCAL CONST Robtarget Tr_meulage_motif_1_P332 :=[[108.4913984375,-190.030578125,1.15107263183594],[0.635107748876336,-0.564376918949611,-0.350307497755773,0.394209966502961],[0,0,0,0],[8.999999E+09,8.999999E+09,8.999999E+09,8.999999E+09,8.999999E+09,8.999999E+09]];
	LOCAL CONST Robtarget Tr_meulage_motif_1_P333 :=[[108.0171015625,-190.910953125,1.15108508300781],[0.635107748876336,-0.564376918949611,-0.350307497755773,0.394209966502961],[0,0,0,0],[8.999999E+09,8.999999E+09,8.999999E+09,8.999999E+09,8.999999E+09,8.999999E+09]];
	LOCAL CONST Robtarget Tr_meulage_motif_1_P334 :=[[107.5428125,-191.7913125,1.15109753417969],[0.635107748876336,-0.564376918949611,-0.350307497755773,0.394209966502961],[0,0,0,0],[8.999999E+09,8.999999E+09,8.999999E+09,8.999999E+09,8.999999E+09,8.999999E+09]];
	LOCAL CONST Robtarget Tr_meulage_motif_1_P335 :=[[107.068515625,-192.6716875,1.15110998535156],[0.635107748876336,-0.564376918949611,-0.350307497755773,0.394209966502961],[0,0,0,0],[8.999999E+09,8.999999E+09,8.999999E+09,8.999999E+09,8.999999E+09,8.999999E+09]];
	LOCAL CONST Robtarget Tr_meulage_motif_1_degg1 :=[[115.967835877567,-197.078596451116,-0.0241570221090994],[0.635107748876336,-0.564376918949611,-0.350307497755773,0.394209966502961],[0,0,0,0],[8.999999E+09,8.999999E+09,8.999999E+09,8.999999E+09,8.999999E+09,8.999999E+09]];
	LOCAL CONST Robtarget Tr_meulage_motif_1_degg2 :=[[285.054920676337,-280.809866522324,-22.3542301638617],[0.635107748876336,-0.564376918949611,-0.350307497755773,0.394209966502961],[0,0,0,0],[8.999999E+09,8.999999E+09,8.999999E+09,8.999999E+09,8.999999E+09,8.999999E+09]];
	LOCAL CONST Robtarget Tr_meulage_motif_2_App1 :=[[13.6932887688866,-23.2749287427864,-194.20163902677],[-3.19370360057134E-06,0.00176428802739274,-0.00181018821640207,-0.999996805242986],[0,0,0,0],[8.999999E+09,8.999999E+09,8.999999E+09,8.999999E+09,8.999999E+09,8.999999E+09]];
	LOCAL CONST Robtarget Tr_meulage_motif_2_App2 :=[[13.0228636571943,-22.5870572769831,-4.2040670343463],[-3.19370360057134E-06,0.00176428802739274,-0.00181018821640207,-0.999996805242986],[0,0,0,0],[8.999999E+09,8.999999E+09,8.999999E+09,8.999999E+09,8.999999E+09,8.999999E+09]];
	LOCAL CONST Robtarget Tr_meulage_motif_2_P0 :=[[12.987578125,-22.550853515625,5.79580517578125],[-3.19370360057134E-06,0.00176428802739274,-0.00181018821640207,-0.999996805242986],[0,0,0,0],[8.999999E+09,8.999999E+09,8.999999E+09,8.999999E+09,8.999999E+09,8.999999E+09]];
	LOCAL CONST Robtarget Tr_meulage_motif_2_P1 :=[[13.9801298828125,-22.6726171875,5.79964208984375],[-3.19370360057134E-06,0.00176428802739274,-0.00181018821640207,-0.999996805242986],[0,0,0,0],[8.999999E+09,8.999999E+09,8.999999E+09,8.999999E+09,8.999999E+09,8.999999E+09]];
	LOCAL CONST Robtarget Tr_meulage_motif_2_P2 :=[[14.972681640625,-22.79437890625,5.8034794921875],[-3.19370360057134E-06,0.00176428802739274,-0.00181018821640207,-0.999996805242986],[0,0,0,0],[8.999999E+09,8.999999E+09,8.999999E+09,8.999999E+09,8.999999E+09,8.999999E+09]];
	LOCAL CONST Robtarget Tr_meulage_motif_2_P3 :=[[15.965234375,-22.916142578125,5.80731689453125],[-3.19370360057134E-06,0.00176428802739274,-0.00181018821640207,-0.999996805242986],[0,0,0,0],[8.999999E+09,8.999999E+09,8.999999E+09,8.999999E+09,8.999999E+09,8.999999E+09]];
	LOCAL CONST Robtarget Tr_meulage_motif_2_P4 :=[[16.95778515625,-23.037904296875,5.811154296875],[-3.19370360057134E-06,0.00176428802739274,-0.00181018821640207,-0.999996805242986],[0,0,0,0],[8.999999E+09,8.999999E+09,8.999999E+09,8.999999E+09,8.999999E+09,8.999999E+09]];
	LOCAL CONST Robtarget Tr_meulage_motif_2_P5 :=[[17.950337890625,-23.15966796875,5.81499169921875],[-3.19370360057134E-06,0.00176428802739274,-0.00181018821640207,-0.999996805242986],[0,0,0,0],[8.999999E+09,8.999999E+09,8.999999E+09,8.999999E+09,8.999999E+09,8.999999E+09]];
	LOCAL CONST Robtarget Tr_meulage_motif_2_P6 :=[[18.942888671875,-23.2814296875,5.8188291015625],[-3.19370360057134E-06,0.00176428802739274,-0.00181018821640207,-0.999996805242986],[0,0,0,0],[8.999999E+09,8.999999E+09,8.999999E+09,8.999999E+09,8.999999E+09,8.999999E+09]];
	LOCAL CONST Robtarget Tr_meulage_motif_2_P7 :=[[19.93544140625,-23.40319140625,5.822666015625],[-3.19370360057134E-06,0.00176428802739274,-0.00181018821640207,-0.999996805242986],[0,0,0,0],[8.999999E+09,8.999999E+09,8.999999E+09,8.999999E+09,8.999999E+09,8.999999E+09]];
	LOCAL CONST Robtarget Tr_meulage_motif_2_P8 :=[[20.9279921875,-23.524955078125,5.82650341796875],[-3.19370360057134E-06,0.00176428802739274,-0.00181018821640207,-0.999996805242986],[0,0,0,0],[8.999999E+09,8.999999E+09,8.999999E+09,8.999999E+09,8.999999E+09,8.999999E+09]];
	LOCAL CONST Robtarget Tr_meulage_motif_2_P9 :=[[21.920544921875,-23.646716796875,5.8303408203125],[-3.19370360057134E-06,0.00176428802739274,-0.00181018821640207,-0.999996805242986],[0,0,0,0],[8.999999E+09,8.999999E+09,8.999999E+09,8.999999E+09,8.999999E+09,8.999999E+09]];
	LOCAL CONST Robtarget Tr_meulage_motif_2_P10 :=[[22.91309765625,-23.76848046875,5.83417822265625],[-3.19370360057134E-06,0.00176428802739274,-0.00181018821640207,-0.999996805242986],[0,0,0,0],[8.999999E+09,8.999999E+09,8.999999E+09,8.999999E+09,8.999999E+09,8.999999E+09]];
	LOCAL CONST Robtarget Tr_meulage_motif_2_P11 :=[[23.9056484375,-23.8902421875,5.838015625],[-3.19370360057134E-06,0.00176428802739274,-0.00181018821640207,-0.999996805242986],[0,0,0,0],[8.999999E+09,8.999999E+09,8.999999E+09,8.999999E+09,8.999999E+09,8.999999E+09]];
	LOCAL CONST Robtarget Tr_meulage_motif_2_P12 :=[[24.898201171875,-24.01200390625,5.8418525390625],[-3.19370360057134E-06,0.00176428802739274,-0.00181018821640207,-0.999996805242986],[0,0,0,0],[8.999999E+09,8.999999E+09,8.999999E+09,8.999999E+09,8.999999E+09,8.999999E+09]];
	LOCAL CONST Robtarget Tr_meulage_motif_2_P13 :=[[25.890751953125,-24.133767578125,5.84568994140625],[-3.19370360057134E-06,0.00176428802739274,-0.00181018821640207,-0.999996805242986],[0,0,0,0],[8.999999E+09,8.999999E+09,8.999999E+09,8.999999E+09,8.999999E+09,8.999999E+09]];
	LOCAL CONST Robtarget Tr_meulage_motif_2_P14 :=[[26.8833046875,-24.255529296875,5.84952734375],[-3.19370360057134E-06,0.00176428802739274,-0.00181018821640207,-0.999996805242986],[0,0,0,0],[8.999999E+09,8.999999E+09,8.999999E+09,8.999999E+09,8.999999E+09,8.999999E+09]];
	LOCAL CONST Robtarget Tr_meulage_motif_2_P15 :=[[27.87585546875,-24.37729296875,5.85336474609375],[-3.19370360057134E-06,0.00176428802739274,-0.00181018821640207,-0.999996805242986],[0,0,0,0],[8.999999E+09,8.999999E+09,8.999999E+09,8.999999E+09,8.999999E+09,8.999999E+09]];
	LOCAL CONST Robtarget Tr_meulage_motif_2_P16 :=[[28.868408203125,-24.4990546875,5.8572021484375],[-3.19370360057134E-06,0.00176428802739274,-0.00181018821640207,-0.999996805242986],[0,0,0,0],[8.999999E+09,8.999999E+09,8.999999E+09,8.999999E+09,8.999999E+09,8.999999E+09]];
	LOCAL CONST Robtarget Tr_meulage_motif_2_P17 :=[[29.860958984375,-24.620818359375,5.86103955078125],[-3.19370360057134E-06,0.00176428802739274,-0.00181018821640207,-0.999996805242986],[0,0,0,0],[8.999999E+09,8.999999E+09,8.999999E+09,8.999999E+09,8.999999E+09,8.999999E+09]];
	LOCAL CONST Robtarget Tr_meulage_motif_2_P18 :=[[30.85351171875,-24.742580078125,5.86487646484375],[-3.19370360057134E-06,0.00176428802739274,-0.00181018821640207,-0.999996805242986],[0,0,0,0],[8.999999E+09,8.999999E+09,8.999999E+09,8.999999E+09,8.999999E+09,8.999999E+09]];
	LOCAL CONST Robtarget Tr_meulage_motif_2_P19 :=[[31.8460625,-24.864341796875,5.8687138671875],[-3.19370360057134E-06,0.00176428802739274,-0.00181018821640207,-0.999996805242986],[0,0,0,0],[8.999999E+09,8.999999E+09,8.999999E+09,8.999999E+09,8.999999E+09,8.999999E+09]];
	LOCAL CONST Robtarget Tr_meulage_motif_2_P20 :=[[32.83861328125,-24.98610546875,5.87255126953125],[-3.19370360057134E-06,0.00176428802739274,-0.00181018821640207,-0.999996805242986],[0,0,0,0],[8.999999E+09,8.999999E+09,8.999999E+09,8.999999E+09,8.999999E+09,8.999999E+09]];
	LOCAL CONST Robtarget Tr_meulage_motif_2_P21 :=[[33.83116796875,-25.1078671875,5.876388671875],[-3.19370360057134E-06,0.00176428802739274,-0.00181018821640207,-0.999996805242986],[0,0,0,0],[8.999999E+09,8.999999E+09,8.999999E+09,8.999999E+09,8.999999E+09,8.999999E+09]];
	LOCAL CONST Robtarget Tr_meulage_motif_2_P22 :=[[34.82371875,-25.229630859375,5.88022607421875],[-3.19370360057134E-06,0.00176428802739274,-0.00181018821640207,-0.999996805242986],[0,0,0,0],[8.999999E+09,8.999999E+09,8.999999E+09,8.999999E+09,8.999999E+09,8.999999E+09]];
	LOCAL CONST Robtarget Tr_meulage_motif_2_P23 :=[[35.81626953125,-25.351392578125,5.88406298828125],[-3.19370360057134E-06,0.00176428802739274,-0.00181018821640207,-0.999996805242986],[0,0,0,0],[8.999999E+09,8.999999E+09,8.999999E+09,8.999999E+09,8.999999E+09,8.999999E+09]];
	LOCAL CONST Robtarget Tr_meulage_motif_2_P24 :=[[36.80882421875,-25.47315625,5.887900390625],[-3.19370360057134E-06,0.00176428802739274,-0.00181018821640207,-0.999996805242986],[0,0,0,0],[8.999999E+09,8.999999E+09,8.999999E+09,8.999999E+09,8.999999E+09,8.999999E+09]];
	LOCAL CONST Robtarget Tr_meulage_motif_2_P25 :=[[37.801375,-25.59491796875,5.89173779296875],[-3.19370360057134E-06,0.00176428802739274,-0.00181018821640207,-0.999996805242986],[0,0,0,0],[8.999999E+09,8.999999E+09,8.999999E+09,8.999999E+09,8.999999E+09,8.999999E+09]];
	LOCAL CONST Robtarget Tr_meulage_motif_2_P26 :=[[38.79392578125,-25.7166796875,5.8955751953125],[-3.19370360057134E-06,0.00176428802739274,-0.00181018821640207,-0.999996805242986],[0,0,0,0],[8.999999E+09,8.999999E+09,8.999999E+09,8.999999E+09,8.999999E+09,8.999999E+09]];
	LOCAL CONST Robtarget Tr_meulage_motif_2_P27 :=[[39.7864765625,-25.838443359375,5.89941259765625],[-3.19370360057134E-06,0.00176428802739274,-0.00181018821640207,-0.999996805242986],[0,0,0,0],[8.999999E+09,8.999999E+09,8.999999E+09,8.999999E+09,8.999999E+09,8.999999E+09]];
	LOCAL CONST Robtarget Tr_meulage_motif_2_P28 :=[[40.77903125,-25.960205078125,5.90324951171875],[-3.19370360057134E-06,0.00176428802739274,-0.00181018821640207,-0.999996805242986],[0,0,0,0],[8.999999E+09,8.999999E+09,8.999999E+09,8.999999E+09,8.999999E+09,8.999999E+09]];
	LOCAL CONST Robtarget Tr_meulage_motif_2_P29 :=[[41.77158203125,-26.08196875,5.9070869140625],[-3.19370360057134E-06,0.00176428802739274,-0.00181018821640207,-0.999996805242986],[0,0,0,0],[8.999999E+09,8.999999E+09,8.999999E+09,8.999999E+09,8.999999E+09,8.999999E+09]];
	LOCAL CONST Robtarget Tr_meulage_motif_2_P30 :=[[42.7641328125,-26.20373046875,5.91092431640625],[-3.19370360057134E-06,0.00176428802739274,-0.00181018821640207,-0.999996805242986],[0,0,0,0],[8.999999E+09,8.999999E+09,8.999999E+09,8.999999E+09,8.999999E+09,8.999999E+09]];
	LOCAL CONST Robtarget Tr_meulage_motif_2_P31 :=[[43.75668359375,-26.325494140625,5.91476171875],[-3.19370360057134E-06,0.00176428802739274,-0.00181018821640207,-0.999996805242986],[0,0,0,0],[8.999999E+09,8.999999E+09,8.999999E+09,8.999999E+09,8.999999E+09,8.999999E+09]];
	LOCAL CONST Robtarget Tr_meulage_motif_2_P32 :=[[44.74923828125,-26.447255859375,5.91859912109375],[-3.19370360057134E-06,0.00176428802739274,-0.00181018821640207,-0.999996805242986],[0,0,0,0],[8.999999E+09,8.999999E+09,8.999999E+09,8.999999E+09,8.999999E+09,8.999999E+09]];
